# B&R Automation Studio project CleanChemi_SiteManagementSystem (part 26)

```iecst
		IF gSkid_LR[IdxSkids_LR].VisBool.P101_AUTOCAL_OFF THEN
			gCMD_LR[IdxSkids_LR].Write_P101_AUTOCAL.wP101_AUTOCAL := 1;
			gCMD_LR[IdxSkids_LR].Write_P101_AUTOCAL.Send := TRUE;
			gSkid_LR[IdxSkids_LR].VisBool.P101_AUTOCAL_OFF := FALSE;
		END_IF;

		IF gSkid_LR[IdxSkids_LR].VisBool.P102_AUTOCAL_ON THEN
			gCMD_LR[IdxSkids_LR].Write_P102_AUTOCAL.wP102_AUTOCAL := 2;
			gCMD_LR[IdxSkids_LR].Write_P102_AUTOCAL.Send := TRUE;
			gSkid_LR[IdxSkids_LR].VisBool.P102_AUTOCAL_ON := FALSE;
		END_IF;

		IF gSkid_LR[IdxSkids_LR].VisBool.P102_AUTOCAL_OFF THEN
			gCMD_LR[IdxSkids_LR].Write_P102_AUTOCAL.wP102_AUTOCAL := 1;
			gCMD_LR[IdxSkids_LR].Write_P102_AUTOCAL.Send := TRUE;
			gSkid_LR[IdxSkids_LR].VisBool.P102_AUTOCAL_OFF := FALSE;
		END_IF;

		IF gSkid_LR[IdxSkids_LR].VisBool.P103_AUTOCAL_ON THEN
			gCMD_LR[IdxSkids_LR].Write_P103_AUTOCAL.wP103_AUTOCAL := 2;
			gCMD_LR[IdxSkids_LR].Write_P103_AUTOCAL.Send := TRUE;
			gSkid_LR[IdxSkids_LR].VisBool.P103_AUTOCAL_ON := FALSE;
		END_IF;

		IF gSkid_LR[IdxSkids_LR].VisBool.P103_AUTOCAL_OFF THEN
			gCMD_LR[IdxSkids_LR].Write_P103_AUTOCAL.wP103_AUTOCAL := 1;
			gCMD_LR[IdxSkids_LR].Write_P103_AUTOCAL.Send := TRUE;
			gSkid_LR[IdxSkids_LR].VisBool.P103_AUTOCAL_OFF := FALSE;
		END_IF;

		IF gSkid_LR[IdxSkids_LR].VisBool.P104_AUTOCAL_ON THEN
			gCMD_LR[IdxSkids_LR].Write_P104_AUTOCAL.wP104_AUTOCAL := 2;
			gCMD_LR[IdxSkids_LR].Write_P104_AUTOCAL.Send := TRUE;
			gSkid_LR[IdxSkids_LR].VisBool.P104_AUTOCAL_ON := FALSE;
		END_IF;

		IF gSkid_LR[IdxSkids_LR].VisBool.P104_AUTOCAL_OFF THEN
			gCMD_LR[IdxSkids_LR].Write_P104_AUTOCAL.wP104_AUTOCAL := 1;
			gCMD_LR[IdxSkids_LR].Write_P104_AUTOCAL.Send := TRUE;
			gSkid_LR[IdxSkids_LR].VisBool.P104_AUTOCAL_OFF := FALSE;
		END_IF;

		IF gSkid_LR[IdxSkids_LR].VisBool.P201_AUTOCAL_ON THEN
			gCMD_LR[IdxSkids_LR].Write_P201_AUTOCAL.wP201_AUTOCAL := 2;
			gCMD_LR[IdxSkids_LR].Write_P201_AUTOCAL.Send := TRUE;
			gSkid_LR[IdxSkids_LR].VisBool.P201_AUTOCAL_ON := FALSE;
		END_IF;

		IF gSkid_LR[IdxSkids_LR].VisBool.P201_AUTOCAL_OFF THEN
			gCMD_LR[IdxSkids_LR].Write_P201_AUTOCAL.wP201_AUTOCAL := 1;
			gCMD_LR[IdxSkids_LR].Write_P201_AUTOCAL.Send := TRUE;
			gSkid_LR[IdxSkids_LR].VisBool.P201_AUTOCAL_OFF := FALSE;
		END_IF;

		IF gSkid_LR[IdxSkids_LR].VisBool.P202_AUTOCAL_ON THEN
			gCMD_LR[IdxSkids_LR].Write_P202_AUTOCAL.wP202_AUTOCAL := 2;
			gCMD_LR[IdxSkids_LR].Write_P202_AUTOCAL.Send := TRUE;
			gSkid_LR[IdxSkids_LR].VisBool.P202_AUTOCAL_ON := FALSE;
		END_IF;

		IF gSkid_LR[IdxSkids_LR].VisBool.P202_AUTOCAL_OFF THEN
			gCMD_LR[IdxSkids_LR].Write_P202_AUTOCAL.wP202_AUTOCAL := 1;
			gCMD_LR[IdxSkids_LR].Write_P202_AUTOCAL.Send := TRUE;
			gSkid_LR[IdxSkids_LR].VisBool.P202_AUTOCAL_OFF := FALSE;
		END_IF;

		IF gSkid_LR[IdxSkids_LR].VisBool.P203_AUTOCAL_ON THEN
			gCMD_LR[IdxSkids_LR].Write_P203_AUTOCAL.wP203_AUTOCAL := 2;
			gCMD_LR[IdxSkids_LR].Write_P203_AUTOCAL.Send := TRUE;
			gSkid_LR[IdxSkids_LR].VisBool.P203_AUTOCAL_ON := FALSE;
		END_IF;

		IF gSkid_LR[IdxSkids_LR].VisBool.P203_AUTOCAL_OFF THEN
			gCMD_LR[IdxSkids_LR].Write_P203_AUTOCAL.wP203_AUTOCAL := 1;
			gCMD_LR[IdxSkids_LR].Write_P203_AUTOCAL.Send := TRUE;
			gSkid_LR[IdxSkids_LR].VisBool.P203_AUTOCAL_OFF := FALSE;
		END_IF;

		// AutoFLOW 1 = Off, 2 = On
		IF gSkid_LR[IdxSkids_LR].VisBool.P102_AUTOFLOW_ON THEN
			gCMD_LR[IdxSkids_LR].Write_P102_AUTOFLO_ADPT.wP102_P102_AUTOFLO_ADPT := 2;
			gCMD_LR[IdxSkids_LR].Write_P102_AUTOFLO_ADPT.Send := TRUE;
			gSkid_LR[IdxSkids_LR].VisBool.P102_AUTOFLOW_ON := FALSE;
		END_IF;

		IF gSkid_LR[IdxSkids_LR].VisBool.P102_AUTOFLOW_OFF THEN
			gCMD_LR[IdxSkids_LR].Write_P102_AUTOFLO_ADPT.wP102_P102_AUTOFLO_ADPT := 1;
			gCMD_LR[IdxSkids_LR].Write_P102_AUTOFLO_ADPT.Send := TRUE;
			gSkid_LR[IdxSkids_LR].VisBool.P102_AUTOFLOW_OFF := FALSE;
		END_IF;

		IF gSkid_LR[IdxSkids_LR].VisBool.P103_AUTOFLOW_ON THEN
			gCMD_LR[IdxSkids_LR].Write_P103_AUTOFLO_ADPT.wP103_P103_AUTOFLO_ADPT := 2;
			gCMD_LR[IdxSkids_LR].Write_P103_AUTOFLO_ADPT.Send := TRUE;
			gSkid_LR[IdxSkids_LR].VisBool.P103_AUTOFLOW_ON := FALSE;
		END_IF;

		IF gSkid_LR[IdxSkids_LR].VisBool.P103_AUTOFLOW_OFF THEN
			gCMD_LR[IdxSkids_LR].Write_P103_AUTOFLO_ADPT.wP103_P103_AUTOFLO_ADPT := 1;
			gCMD_LR[IdxSkids_LR].Write_P103_AUTOFLO_ADPT.Send := TRUE;
			gSkid_LR[IdxSkids_LR].VisBool.P103_AUTOFLOW_OFF := FALSE;
		END_IF;

		IF gSkid_LR[IdxSkids_LR].VisBool.P104_AUTOFLOW_ON THEN
			gCMD_LR[IdxSkids_LR].Write_P104_AUTOFLO_ADPT.wP104_P104_AUTOFLO_ADPT := 2;
			gCMD_LR[IdxSkids_LR].Write_P104_AUTOFLO_ADPT.Send := TRUE;
			gSkid_LR[IdxSkids_LR].VisBool.P104_AUTOFLOW_ON := FALSE;
		END_IF;

		IF gSkid_LR[IdxSkids_LR].VisBool.P104_AUTOFLOW_OFF THEN
			gCMD_LR[IdxSkids_LR].Write_P104_AUTOFLO_ADPT.wP104_P104_AUTOFLO_ADPT := 1;
			gCMD_LR[IdxSkids_LR].Write_P104_AUTOFLO_ADPT.Send := TRUE;
			gSkid_LR[IdxSkids_LR].VisBool.P104_AUTOFLOW_OFF := FALSE;
		END_IF;

		IF gSkid_LR[IdxSkids_LR].VisBool.P201_AUTOFLOW_ON THEN
			gCMD_LR[IdxSkids_LR].Write_P201_AUTOFLO_ADPT.wP201_P201_AUTOFLO_ADPT := 2;
			gCMD_LR[IdxSkids_LR].Write_P201_AUTOFLO_ADPT.Send := TRUE;
			gSkid_LR[IdxSkids_LR].VisBool.P201_AUTOFLOW_ON := FALSE;
		END_IF;

		IF gSkid_LR[IdxSkids_LR].VisBool.P201_AUTOFLOW_OFF THEN
			gCMD_LR[IdxSkids_LR].Write_P201_AUTOFLO_ADPT.wP201_P201_AUTOFLO_ADPT := 1;
			gCMD_LR[IdxSkids_LR].Write_P201_AUTOFLO_ADPT.Send := TRUE;
			gSkid_LR[IdxSkids_LR].VisBool.P201_AUTOFLOW_OFF := FALSE;
		END_IF;

		IF gSkid_LR[IdxSkids_LR].VisBool.P202_AUTOFLOW_ON THEN
			gCMD_LR[IdxSkids_LR].Write_P202_AUTOFLO_ADPT.wP202_P202_AUTOFLO_ADPT := 2;
			gCMD_LR[IdxSkids_LR].Write_P202_AUTOFLO_ADPT.Send := TRUE;
			gSkid_LR[IdxSkids_LR].VisBool.P202_AUTOFLOW_ON := FALSE;
		END_IF;

		IF gSkid_LR[IdxSkids_LR].VisBool.P202_AUTOFLOW_OFF THEN
			gCMD_LR[IdxSkids_LR].Write_P202_AUTOFLO_ADPT.wP202_P202_AUTOFLO_ADPT := 1;
			gCMD_LR[IdxSkids_LR].Write_P202_AUTOFLO_ADPT.Send := TRUE;
			gSkid_LR[IdxSkids_LR].VisBool.P202_AUTOFLOW_OFF := FALSE;
		END_IF;

		IF gSkid_LR[IdxSkids_LR].VisBool.P203_AUTOFLOW_ON THEN
			gCMD_LR[IdxSkids_LR].Write_P203_AUTOFLO_ADPT.wP203_P203_AUTOFLO_ADPT := 2;
			gCMD_LR[IdxSkids_LR].Write_P203_AUTOFLO_ADPT.Send := TRUE;
			gSkid_LR[IdxSkids_LR].VisBool.P203_AUTOFLOW_ON := FALSE;
		END_IF;

		IF gSkid_LR[IdxSkids_LR].VisBool.P203_AUTOFLOW_OFF THEN
			gCMD_LR[IdxSkids_LR].Write_P203_AUTOFLO_ADPT.wP203_P203_AUTOFLO_ADPT := 1;
			gCMD_LR[IdxSkids_LR].Write_P203_AUTOFLO_ADPT.Send := TRUE;
			gSkid_LR[IdxSkids_LR].VisBool.P203_AUTOFLOW_OFF := FALSE;
		END_IF;

		// Autocal PV 1 = FIT, 2 = PFIT
		IF gSkid_LR[IdxSkids_LR].VisBool.P104_PV_FIT THEN
			gCMD_LR[IdxSkids_LR].Write_P104_AUTOCAL_PV.wP104_AUTOCAL_PV := 1;
			gCMD_LR[IdxSkids_LR].Write_P104_AUTOCAL_PV.Send := TRUE;
			gSkid_LR[IdxSkids_LR].VisBool.P104_PV_FIT := FALSE;
		END_IF;

		IF gSkid_LR[IdxSkids_LR].VisBool.P104_PV_PFIT THEN
			gCMD_LR[IdxSkids_LR].Write_P104_AUTOCAL_PV.wP104_AUTOCAL_PV := 2;
			gCMD_LR[IdxSkids_LR].Write_P104_AUTOCAL_PV.Send := TRUE;
			gSkid_LR[IdxSkids_LR].VisBool.P104_PV_PFIT := FALSE;
		END_IF;

		IF gSkid_LR[IdxSkids_LR].VisBool.P201_PV_FIT THEN
			gCMD_LR[IdxSkids_LR].Write_P201_AUTOCAL_PV.wP201_AUTOCAL_PV := 1;
			gCMD_LR[IdxSkids_LR].Write_P201_AUTOCAL_PV.Send := TRUE;
			gSkid_LR[IdxSkids_LR].VisBool.P201_PV_FIT := FALSE;
		END_IF;

		IF gSkid_LR[IdxSkids_LR].VisBool.P201_PV_PFIT THEN
			gCMD_LR[IdxSkids_LR].Write_P201_AUTOCAL_PV.wP201_AUTOCAL_PV := 2;
			gCMD_LR[IdxSkids_LR].Write_P201_AUTOCAL_PV.Send := TRUE;
			gSkid_LR[IdxSkids_LR].VisBool.P201_PV_PFIT := FALSE;
		END_IF;

		IF gSkid_LR[IdxSkids_LR].VisBool.P202_PV_FIT THEN
			gCMD_LR[IdxSkids_LR].Write_P202_AUTOCAL_PV.wP202_AUTOCAL_PV := 1;
			gCMD_LR[IdxSkids_LR].Write_P202_AUTOCAL_PV.Send := TRUE;
			gSkid_LR[IdxSkids_LR].VisBool.P202_PV_FIT := FALSE;
		END_IF;

		IF gSkid_LR[IdxSkids_LR].VisBool.P202_PV_PFIT THEN
			gCMD_LR[IdxSkids_LR].Write_P202_AUTOCAL_PV.wP202_AUTOCAL_PV := 2;
			gCMD_LR[IdxSkids_LR].Write_P202_AUTOCAL_PV.Send := TRUE;
			gSkid_LR[IdxSkids_LR].VisBool.P202_PV_PFIT := FALSE;
		END_IF;

		IF gSkid_LR[IdxSkids_LR].VisBool.P203_PV_FIT THEN
			gCMD_LR[IdxSkids_LR].Write_P203_AUTOCAL_PV.wP203_AUTOCAL_PV := 1;
			gCMD_LR[IdxSkids_LR].Write_P203_AUTOCAL_PV.Send := TRUE;
			gSkid_LR[IdxSkids_LR].VisBool.P203_PV_FIT := FALSE;
		END_IF;

		IF gSkid_LR[IdxSkids_LR].VisBool.P203_PV_PFIT THEN
			gCMD_LR[IdxSkids_LR].Write_P203_AUTOCAL_PV.wP203_AUTOCAL_PV := 2;
			gCMD_LR[IdxSkids_LR].Write_P203_AUTOCAL_PV.Send := TRUE;
			gSkid_LR[IdxSkids_LR].VisBool.P203_PV_PFIT := FALSE;
		END_IF;

		gSkid_LR[IdxSkids_LR].BufferTank.LI200P := (gSkid_LR[IdxSkids_LR].BufferTank.LI200 / BT_VOLUME)*100;

		gSkid_LR[IdxSkids_LR].VisBool.CD101_TARGETHI := gSkid_LR[IdxSkids_LR].Sensor_Variables.CD101_SP + 40;
		gSkid_LR[IdxSkids_LR].VisBool.CD101_TARGETLO := gSkid_LR[IdxSkids_LR].Sensor_Variables.CD101_SP - 40;
		gSkid_LR[IdxSkids_LR].VisBool.CD102_TARGETHI := gSkid_LR[IdxSkids_LR].Sensor_Variables.CD102_SP + 40;
		gSkid_LR[IdxSkids_LR].VisBool.CD102_TARGETLO := gSkid_LR[IdxSkids_LR].Sensor_Variables.CD102_SP - 40;

		// VISIBILITY TRIGGER SETTING

		IF gSkid_LR[IdxSkids_LR].BufferTank.LSHH200 > LSHH200_TRIGGER THEN
			gSkid_LR[IdxSkids_LR].VisBool.LSHH200 := 1;
		ELSE
			gSkid_LR[IdxSkids_LR].VisBool.LSHH200 := 0;
		END_IF;

		IF gSkid_LR[IdxSkids_LR].Pmax_Pump_102.P102_LS > P102_LS_TRIGGER THEN
			gSkid_LR[IdxSkids_LR].VisBool.P102_LS := 1;
		ELSE
			gSkid_LR[IdxSkids_LR].VisBool.P102_LS := 0;
		END_IF;

		IF gSkid_LR[IdxSkids_LR].Pmax_Pump_103.P103_LS > P103_LS_TRIGGER THEN
			gSkid_LR[IdxSkids_LR].VisBool.P103_LS := 1;
		ELSE
			gSkid_LR[IdxSkids_LR].VisBool.P103_LS := 0;
		END_IF;

		IF gSkid_LR[IdxSkids_LR].Pmax_General_Variables.PMAX_HOA = 2 THEN
			gSkid_LR[IdxSkids_LR].VisBool.PMAX_MANUAL := 1;
		ELSE
			gSkid_LR[IdxSkids_LR].VisBool.PMAX_MANUAL := 0;
		END_IF;

		IF gSkid_LR[IdxSkids_LR].Dosing_Pump_201.P201_HOA = 0 OR gSkid_LR[IdxSkids_LR].Dosing_Pump_201.P201_HOA = 8  THEN
			gSkid_LR[IdxSkids_LR].VisBool.P201_PPM := 0;
		ELSE
			gSkid_LR[IdxSkids_LR].VisBool.P201_PPM := 1;
		END_IF;

		IF gSkid_LR[IdxSkids_LR].Dosing_Pump_202.P202_HOA = 0 OR gSkid_LR[IdxSkids_LR].Dosing_Pump_202.P202_HOA = 8  THEN
			gSkid_LR[IdxSkids_LR].VisBool.P202_PPM := 0;
		ELSE
			gSkid_LR[IdxSkids_LR].VisBool.P202_PPM := 1;
		END_IF;

		IF gSkid_LR[IdxSkids_LR].Dosing_Pump_203.P203_HOA = 0 OR gSkid_LR[IdxSkids_LR].Dosing_Pump_203.P203_HOA = 8  THEN
			gSkid_LR[IdxSkids_LR].VisBool.P203_PPM := 0;
		ELSE
			gSkid_LR[IdxSkids_LR].VisBool.P203_PPM := 1;
		END_IF;

		IF gSkid_LR[IdxSkids_LR].Dosing_Pump_201.P201_HOA = 8 THEN
			gSkid_LR[IdxSkids_LR].VisBool.P201_SP := 1;
		ELSE
			gSkid_LR[IdxSkids_LR].VisBool.P201_SP := 0;
		END_IF;

		IF gSkid_LR[IdxSkids_LR].Dosing_Pump_202.P202_HOA = 8 THEN
			gSkid_LR[IdxSkids_LR].VisBool.P202_SP := 1;
		ELSE
			gSkid_LR[IdxSkids_LR].VisBool.P202_SP := 0;
		END_IF;

		IF gSkid_LR[IdxSkids_LR].Dosing_Pump_203.P203_HOA = 8 THEN
			gSkid_LR[IdxSkids_LR].VisBool.P203_SP := 1;
		ELSE
			gSkid_LR[IdxSkids_LR].VisBool.P203_SP := 0;
		END_IF;

		IF gSkid_LR[IdxSkids_LR].Dosing_Pump_201.P201_ENABLE = 1 THEN
			gSkid_LR[IdxSkids_LR].VisBool.P201_ENABLE_OPP := 0;
		ELSE
			gSkid_LR[IdxSkids_LR].VisBool.P201_ENABLE_OPP := 1;
		END_IF;

		IF gSkid_LR[IdxSkids_LR].Dosing_Pump_202.P202_ENABLE = 1 THEN
			gSkid_LR[IdxSkids_LR].VisBool.P202_ENABLE_OPP := 0;
		ELSE
			gSkid_LR[IdxSkids_LR].VisBool.P202_ENABLE_OPP := 1;
		END_IF;

		IF gSkid_LR[IdxSkids_LR].Dosing_Pump_203.P203_ENABLE = 1 THEN
			gSkid_LR[IdxSkids_LR].VisBool.P203_ENABLE_OPP := 0;
		ELSE
			gSkid_LR[IdxSkids_LR].VisBool.P203_ENABLE_OPP := 1;
		END_IF;

		IF gSkid_LR[IdxSkids_LR].Pmax_Pump_102.P102_WARN > 0 THEN
			gSkid_LR[IdxSkids_LR].VisBool.P102_WARN := 1;
		ELSE
			gSkid_LR[IdxSkids_LR].VisBool.P102_WARN := 0;
		END_IF;

		IF gSkid_LR[IdxSkids_LR].Pmax_Pump_102.P102_ALARM > 0 THEN
			gSkid_LR[IdxSkids_LR].VisBool.P102_ALARM := 1;
		ELSE
			gSkid_LR[IdxSkids_LR].VisBool.P102_ALARM := 0;
		END_IF;

		IF gSkid_LR[IdxSkids_LR].Pmax_Pump_103.P103_WARN > 0 THEN
			gSkid_LR[IdxSkids_LR].VisBool.P103_WARN := 1;
		ELSE
			gSkid_LR[IdxSkids_LR].VisBool.P103_WARN := 0;
		END_IF;

		IF gSkid_LR[IdxSkids_LR].Pmax_Pump_103.P103_ALARM > 0 THEN
			gSkid_LR[IdxSkids_LR].VisBool.P103_ALARM := 1;
		ELSE
			gSkid_LR[IdxSkids_LR].VisBool.P103_ALARM := 0;
		END_IF;

		IF gSkid_LR[IdxSkids_LR].Pmax_Pump_104.P104_WARN > 0 THEN
			gSkid_LR[IdxSkids_LR].VisBool.P104_WARN := 1;
		ELSE
			gSkid_LR[IdxSkids_LR].VisBool.P104_WARN := 0;
		END_IF;

		IF gSkid_LR[IdxSkids_LR].Pmax_Pump_104.P104_ALARM > 0 THEN
			gSkid_LR[IdxSkids_LR].VisBool.P104_ALARM := 1;
		ELSE
			gSkid_LR[IdxSkids_LR].VisBool.P104_ALARM := 0;
		END_IF;

		IF gSkid_LR[IdxSkids_LR].Dosing_Pump_201.P201_WARN > 0 AND gSkid_LR[IdxSkids_LR].VisBool.P201_DME = 0 THEN
			gSkid_LR[IdxSkids_LR].VisBool.P201_WARN := 1;
		ELSE
			gSkid_LR[IdxSkids_LR].VisBool.P201_WARN := 0;
		END_IF;

		IF gSkid_LR[IdxSkids_LR].Dosing_Pump_201.P201_ALARM > 0 AND gSkid_LR[IdxSkids_LR].VisBool.P201_DME = 0  THEN
			gSkid_LR[IdxSkids_LR].VisBool.P201_ALARM := 1;
		ELSE
			gSkid_LR[IdxSkids_LR].VisBool.P201_ALARM := 0;
		END_IF;

		IF gSkid_LR[IdxSkids_LR].Dosing_Pump_202.P202_WARN > 0 THEN
			gSkid_LR[IdxSkids_LR].VisBool.P202_WARN := 1;
		ELSE
			gSkid_LR[IdxSkids_LR].VisBool.P202_WARN := 0;
		END_IF;

		IF gSkid_LR[IdxSkids_LR].Dosing_Pump_202.P202_ALARM > 0 THEN
			gSkid_LR[IdxSkids_LR].VisBool.P202_ALARM := 1;
		ELSE
			gSkid_LR[IdxSkids_LR].VisBool.P202_ALARM := 0;
		END_IF;

		IF gSkid_LR[IdxSkids_LR].Dosing_Pump_203.P203_WARN > 0 THEN
			gSkid_LR[IdxSkids_LR].VisBool.P203_WARN := 1;
		ELSE
			gSkid_LR[IdxSkids_LR].VisBool.P203_WARN := 0;
		END_IF;

		IF gSkid_LR[IdxSkids_LR].Dosing_Pump_203.P203_ALARM > 0 THEN
			gSkid_LR[IdxSkids_LR].VisBool.P203_ALARM := 1;
		ELSE
			gSkid_LR[IdxSkids_LR].VisBool.P203_ALARM := 0;
		END_IF;

		IF gSkid_LR[IdxSkids_LR].Dosing_Pump_201.P201_ADJ = 1 AND gSkid_LR[IdxSkids_LR].VisBool.P201_PPM = 1 THEN
			gSkid_LR[IdxSkids_LR].VisBool.P201_APPM := 1;
		ELSE
			gSkid_LR[IdxSkids_LR].VisBool.P201_APPM := 0;
		END_IF;

		IF gSkid_LR[IdxSkids_LR].Dosing_Pump_202.P202_ADJ = 1 AND gSkid_LR[IdxSkids_LR].VisBool.P202_PPM = 1 THEN
			gSkid_LR[IdxSkids_LR].VisBool.P202_APPM := 1;
		ELSE
			gSkid_LR[IdxSkids_LR].VisBool.P202_APPM := 0;
		END_IF;

		IF gSkid_LR[IdxSkids_LR].Dosing_Pump_203.P203_ADJ = 1 AND gSkid_LR[IdxSkids_LR].VisBool.P203_PPM = 1 THEN
			gSkid_LR[IdxSkids_LR].VisBool.P203_APPM := 1;
		ELSE
			gSkid_LR[IdxSkids_LR].VisBool.P203_APPM := 0;
		END_IF;

		IF gSkid_LR[IdxSkids_LR].Sensor_Variables.FI301_MODE = 0 AND gSkid_LR[IdxSkids_LR].Pmax_General_Variables.SCREEN_LOCK = 1 THEN
			gSkid_LR[IdxSkids_LR].VisBool.FI301_MODE_OPP := 1;
		ELSE
			gSkid_LR[IdxSkids_LR].VisBool.FI301_MODE_OPP := 0;
		END_IF;

		IF gSkid_LR[IdxSkids_LR].Sensor_Variables.FI302_MODE = 0 AND gSkid_LR[IdxSkids_LR].Pmax_General_Variables.SCREEN_LOCK = 1 THEN
			gSkid_LR[IdxSkids_LR].VisBool.FI302_MODE_OPP := 1;
		ELSE
			gSkid_LR[IdxSkids_LR].VisBool.FI302_MODE_OPP := 0;
		END_IF;

		IF gSkid_LR[IdxSkids_LR].Sensor_Variables.FI303_MODE = 0 AND gSkid_LR[IdxSkids_LR].Pmax_General_Variables.SCREEN_LOCK = 1 THEN
			gSkid_LR[IdxSkids_LR].VisBool.FI303_MODE_OPP := 1;
		ELSE
			gSkid_LR[IdxSkids_LR].VisBool.FI303_MODE_OPP := 0;
		END_IF;

		IF gSkid_LR[IdxSkids_LR].Sensor_Variables.FI301_MODE = 1 AND gSkid_LR[IdxSkids_LR].Pmax_General_Variables.SCREEN_LOCK = 1 THEN
			gSkid_LR[IdxSkids_LR].VisBool.FI301_MODE := 1;
		ELSE
			gSkid_LR[IdxSkids_LR].VisBool.FI301_MODE := 0;
		END_IF;

		IF gSkid_LR[IdxSkids_LR].Sensor_Variables.FI302_MODE = 1 AND gSkid_LR[IdxSkids_LR].Pmax_General_Variables.SCREEN_LOCK = 1 THEN
			gSkid_LR[IdxSkids_LR].VisBool.FI302_MODE := 1;
		ELSE
			gSkid_LR[IdxSkids_LR].VisBool.FI302_MODE := 0;
		END_IF;

		IF gSkid_LR[IdxSkids_LR].Sensor_Variables.FI303_MODE = 1 AND gSkid_LR[IdxSkids_LR].Pmax_General_Variables.SCREEN_LOCK = 1 THEN
			gSkid_LR[IdxSkids_LR].VisBool.FI303_MODE := 1;
		ELSE
			gSkid_LR[IdxSkids_LR].VisBool.FI303_MODE := 0;
		END_IF;

		IF gSkid_LR[IdxSkids_LR].Sensor_Variables.XV101 = 0 AND gSkid_LR[IdxSkids_LR].Sensor_Variables.XV101_ENABLE = 1 THEN
			gSkid_LR[IdxSkids_LR].VisBool.XV101_OPP := 1;
		ELSE
			gSkid_LR[IdxSkids_LR].VisBool.XV101_OPP := 0;
		END_IF;

		IF gSkid_LR[IdxSkids_LR].Sensor_Variables.XV101 = 2 AND gSkid_LR[IdxSkids_LR].Sensor_Variables.XV101_ENABLE = 1 THEN
			gSkid_LR[IdxSkids_LR].VisBool.XV101_ERROR := 1;
		ELSE
			gSkid_LR[IdxSkids_LR].VisBool.XV101_ERROR := 0;
		END_IF;

		IF gSkid_LR[IdxSkids_LR].Sensor_Variables.XV101 = 1 AND gSkid_LR[IdxSkids_LR].Sensor_Variables.XV101_ENABLE = 1 THEN
			gSkid_LR[IdxSkids_LR].VisBool.XV101 := 1;
		ELSE
			gSkid_LR[IdxSkids_LR].VisBool.XV101 := 0;
		END_IF;

		IF gSkid_LR[IdxSkids_LR].Sensor_Variables.XV102 = 0 AND gSkid_LR[IdxSkids_LR].Pmax_Pump_102.XV102_ENABLE = 1 THEN
			gSkid_LR[IdxSkids_LR].VisBool.XV102_OPP := 1;
		ELSE
			gSkid_LR[IdxSkids_LR].VisBool.XV102_OPP := 0;
		END_IF;

		IF gSkid_LR[IdxSkids_LR].Sensor_Variables.XV102 = 1 AND gSkid_LR[IdxSkids_LR].Pmax_Pump_102.XV102_ENABLE = 1 THEN
			gSkid_LR[IdxSkids_LR].VisBool.XV102 := 1;
		ELSE
			gSkid_LR[IdxSkids_LR].VisBool.XV102 := 0;
		END_IF;

		IF gSkid_LR[IdxSkids_LR].Sensor_Variables.XV103 = 1 THEN
			gSkid_LR[IdxSkids_LR].VisBool.XV103_OPP := 0;
		ELSE
			gSkid_LR[IdxSkids_LR].VisBool.XV103_OPP := 1;
		END_IF;

		IF gSkid_LR[IdxSkids_LR].Sensor_Variables.XV104 = 0 AND gSkid_LR[IdxSkids_LR].Pmax_Pump_104.XV104_ENABLE = 1 THEN
			gSkid_LR[IdxSkids_LR].VisBool.XV104_OPP := 1;
		ELSE
			gSkid_LR[IdxSkids_LR].VisBool.XV104_OPP := 0;
		END_IF;

		IF gSkid_LR[IdxSkids_LR].Sensor_Variables.XV104 = 1 AND gSkid_LR[IdxSkids_LR].Pmax_Pump_104.XV104_ENABLE = 1 THEN
			gSkid_LR[IdxSkids_LR].VisBool.XV104 := 1;
		ELSE
			gSkid_LR[IdxSkids_LR].VisBool.XV104 := 0;
		END_IF;

		IF gSkid_LR[IdxSkids_LR].Sensor_Variables.XV201 = 1 THEN
			gSkid_LR[IdxSkids_LR].VisBool.XV201_OPP := 0;
		ELSE
			gSkid_LR[IdxSkids_LR].VisBool.XV201_OPP := 1;
		END_IF;

		IF gSkid_LR[IdxSkids_LR].Sensor_Variables.XV202 = 1 THEN
			gSkid_LR[IdxSkids_LR].VisBool.XV202_OPP := 0;
		ELSE
			gSkid_LR[IdxSkids_LR].VisBool.XV202_OPP := 1;
		END_IF;

		IF gSkid_LR[IdxSkids_LR].Sensor_Variables.XV203 = 1 THEN
			gSkid_LR[IdxSkids_LR].VisBool.XV203_OPP := 0;
		ELSE
			gSkid_LR[IdxSkids_LR].VisBool.XV203_OPP := 1;
		END_IF;

		IF gSkid_LR[IdxSkids_LR].Dosing_Pump_201.P201_PTYPE = 1 THEN
			gSkid_LR[IdxSkids_LR].VisBool.P201_PTYPE_OPP := 0;
		ELSE
			gSkid_LR[IdxSkids_LR].VisBool.P201_PTYPE_OPP := 1;
		END_IF;

		IF gSkid_LR[IdxSkids_LR].Pmax_General_Variables.SCREEN_LOCK = 1 AND gSkid_LR[IdxSkids_LR].Pmax_General_Variables.PMAX_HOA = 2 THEN
			gSkid_LR[IdxSkids_LR].VisBool.P101_MODE := 1;
			gSkid_LR[IdxSkids_LR].VisBool.P102_MODE := 1;
			gSkid_LR[IdxSkids_LR].VisBool.P103_MODE := 1;
			gSkid_LR[IdxSkids_LR].VisBool.P104_MODE := 1;
		ELSE
			gSkid_LR[IdxSkids_LR].VisBool.P101_MODE := 0;
			gSkid_LR[IdxSkids_LR].VisBool.P102_MODE := 0;
			gSkid_LR[IdxSkids_LR].VisBool.P103_MODE := 0;
			gSkid_LR[IdxSkids_LR].VisBool.P104_MODE := 0;
		END_IF;

		IF gSkid_LR[IdxSkids_LR].Pmax_General_Variables.SCREEN_LOCK = 1 AND gSkid_LR[IdxSkids_LR].Dosing_Pump_201.P201_HOA = 8 THEN
			gSkid_LR[IdxSkids_LR].VisBool.P201_MODE := 1;
		ELSE
			gSkid_LR[IdxSkids_LR].VisBool.P201_MODE := 0;
		END_IF;

		IF gSkid_LR[IdxSkids_LR].Pmax_General_Variables.SCREEN_LOCK = 1 AND gSkid_LR[IdxSkids_LR].Dosing_Pump_202.P202_HOA = 8 THEN
			gSkid_LR[IdxSkids_LR].VisBool.P202_MODE := 1;
		ELSE
			gSkid_LR[IdxSkids_LR].VisBool.P202_MODE := 0;
		END_IF;

		IF gSkid_LR[IdxSkids_LR].Pmax_General_Variables.SCREEN_LOCK = 1 AND gSkid_LR[IdxSkids_LR].Dosing_Pump_203.P203_HOA = 8 THEN
			gSkid_LR[IdxSkids_LR].VisBool.P203_MODE := 1;
		ELSE
			gSkid_LR[IdxSkids_LR].VisBool.P203_MODE := 0;
		END_IF;

		IF gSkid_LR[IdxSkids_LR].Heartbeat.SYSTEM_OFFLINE = 1 THEN
			gSkid_LR[IdxSkids_LR].VisBool.IOSTATUS := 1;
		ELSE
			gSkid_LR[IdxSkids_LR].VisBool.IOSTATUS := 0;
		END_IF;

		//P101 Pump Graphic Vis
		IF gSkid_LR[IdxSkids_LR].Pmax_Pump_101.P101_XS = 1 THEN
			gSkid_LR[IdxSkids_LR].VisBool.P101_DMEYELLOW := 1;
		ELSE
			gSkid_LR[IdxSkids_LR].VisBool.P101_DMEYELLOW := 0;
		END_IF;

		IF gSkid_LR[IdxSkids_LR].Pmax_Pump_101.P101_XS = 3 THEN
			gSkid_LR[IdxSkids_LR].VisBool.P101_DMEGREEN := 1;
		ELSE
			gSkid_LR[IdxSkids_LR].VisBool.P101_DMEGREEN := 0;
		END_IF;

		//P102 Pump Graphic Vis
		IF gSkid_LR[IdxSkids_LR].Pmax_Pump_102.P102_XS = 1 THEN
			gSkid_LR[IdxSkids_LR].VisBool.P102_DDAYELLOW := 1;
		ELSE
			gSkid_LR[IdxSkids_LR].VisBool.P102_DDAYELLOW := 0;
		END_IF;

		IF gSkid_LR[IdxSkids_LR].Pmax_Pump_102.P102_XS = 3 THEN
			gSkid_LR[IdxSkids_LR].VisBool.P102_DDAGREEN := 1;
		ELSE
			gSkid_LR[IdxSkids_LR].VisBool.P102_DDAGREEN := 0;
		END_IF;

		//P103 Pump Graphic Vis
		IF gSkid_LR[IdxSkids_LR].Pmax_Pump_103.P103_XS = 1 THEN
			gSkid_LR[IdxSkids_LR].VisBool.P103_DDAYELLOW := 1;
		ELSE
			gSkid_LR[IdxSkids_LR].VisBool.P103_DDAYELLOW := 0;
		END_IF;

		IF gSkid_LR[IdxSkids_LR].Pmax_Pump_103.P103_XS = 3 THEN
			gSkid_LR[IdxSkids_LR].VisBool.P103_DDAGREEN := 1;
		ELSE
			gSkid_LR[IdxSkids_LR].VisBool.P103_DDAGREEN := 0;
		END_IF;

		//P104 Pump Graphic Vis
		IF gSkid_LR[IdxSkids_LR].Pmax_Pump_104.P104_XS = 1 THEN
			gSkid_LR[IdxSkids_LR].VisBool.P104_DDAYELLOW := 1;
		ELSE
			gSkid_LR[IdxSkids_LR].VisBool.P104_DDAYELLOW := 0;
		END_IF;

		IF gSkid_LR[IdxSkids_LR].Pmax_Pump_104.P104_XS = 3 THEN
			gSkid_LR[IdxSkids_LR].VisBool.P104_DDAGREEN := 1;
		ELSE
			gSkid_LR[IdxSkids_LR].VisBool.P104_DDAGREEN := 0;
		END_IF;

		//P201 Pump Graphic Vis
		IF gSkid_LR[IdxSkids_LR].Dosing_Pump_201.P201_PTYPE = 0 THEN
			gSkid_LR[IdxSkids_LR].VisBool.P201_DDA := 1;
			gSkid_LR[IdxSkids_LR].VisBool.P201_DME := 0;
		ELSE
			gSkid_LR[IdxSkids_LR].VisBool.P201_DDA := 0;
			gSkid_LR[IdxSkids_LR].VisBool.P201_DME := 1;
		END_IF;

		IF gSkid_LR[IdxSkids_LR].Dosing_Pump_201.P201_PTYPE = 1 AND gSkid_LR[IdxSkids_LR].Dosing_Pump_201.P201_XS = 3 THEN
			gSkid_LR[IdxSkids_LR].VisBool.P201_DMEGREEN := 1;
		ELSE
			gSkid_LR[IdxSkids_LR].VisBool.P201_DMEGREEN := 0;
		END_IF;

		IF gSkid_LR[IdxSkids_LR].Dosing_Pump_201.P201_PTYPE = 1 AND gSkid_LR[IdxSkids_LR].Dosing_Pump_201.P201_XS = 1 THEN
			gSkid_LR[IdxSkids_LR].VisBool.P201_DMEYELLOW := 1;
		ELSE
			gSkid_LR[IdxSkids_LR].VisBool.P201_DMEYELLOW := 0;
		END_IF;

		IF gSkid_LR[IdxSkids_LR].Dosing_Pump_201.P201_XS = 1 AND gSkid_LR[IdxSkids_LR].Dosing_Pump_201.P201_PTYPE = 0 THEN
			gSkid_LR[IdxSkids_LR].VisBool.P201_DDAYELLOW := 1;
		ELSE
			gSkid_LR[IdxSkids_LR].VisBool.P201_DDAYELLOW := 0;
		END_IF;

		IF gSkid_LR[IdxSkids_LR].Dosing_Pump_201.P201_XS = 3 AND gSkid_LR[IdxSkids_LR].Dosing_Pump_201.P201_PTYPE = 0 THEN
			gSkid_LR[IdxSkids_LR].VisBool.P201_DDAGREEN := 1;
		ELSE
			gSkid_LR[IdxSkids_LR].VisBool.P201_DDAGREEN := 0;
		END_IF;

		//P202 Pump Graphic Vis
		IF gSkid_LR[IdxSkids_LR].Dosing_Pump_202.P202_XS = 1 THEN
			gSkid_LR[IdxSkids_LR].VisBool.P202_DDAYELLOW := 1;
		ELSE
			gSkid_LR[IdxSkids_LR].VisBool.P202_DDAYELLOW := 0;
		END_IF;

		IF gSkid_LR[IdxSkids_LR].Dosing_Pump_202.P202_XS = 3 THEN
			gSkid_LR[IdxSkids_LR].VisBool.P202_DDAGREEN := 1;
		ELSE
			gSkid_LR[IdxSkids_LR].VisBool.P202_DDAGREEN := 0;
		END_IF;

		//P203 Pump Graphic Vis
		IF gSkid_LR[IdxSkids_LR].Dosing_Pump_203.P203_XS = 1 THEN
			gSkid_LR[IdxSkids_LR].VisBool.P203_DDAYELLOW := 1;
		ELSE
			gSkid_LR[IdxSkids_LR].VisBool.P203_DDAYELLOW := 0;
		END_IF;

		IF gSkid_LR[IdxSkids_LR].Dosing_Pump_203.P203_XS = 3 THEN
			gSkid_LR[IdxSkids_LR].VisBool.P203_DDAGREEN := 1;
		ELSE
			gSkid_LR[IdxSkids_LR].VisBool.P203_DDAGREEN := 0;
		END_IF;

	END_FOR;

END_ACTION
```

#### Main_HR.st
```iecst
ACTION Vis_Main_HR:

	FOR IdxSkids_HR := 0 TO MAX_SKIDS_HR DO

		gSkid_HR[IdxSkids_HR].BufferTank.LI200P := (gSkid_HR[IdxSkids_HR].BufferTank.LI200 / BT_VOLUME)*100;

		// VISIBILITY TRIGGER SETTING

		IF gSkid_LR[IdxSkids_HR].Pmax_General_Variables.HEARTBEAT = 1 THEN
			gSkid_LR[IdxSkids_HR].VisBool.HEARTBEAT := 0;
		ELSE
			gSkid_LR[IdxSkids_HR].VisBool.HEARTBEAT := 1;
		END_IF;

		IF gSkid_HR[IdxSkids_HR].BufferTank.LSHH200 > LSHH200_TRIGGER THEN
			gSkid_HR[IdxSkids_HR].VisBool.LSHH200 := 1;
		ELSE
			gSkid_HR[IdxSkids_HR].VisBool.LSHH200 := 0;
		END_IF;

		IF gSkid_HR[IdxSkids_HR].Pmax_Pump_102.P102_LS > P102_LS_TRIGGER THEN
			gSkid_HR[IdxSkids_HR].VisBool.P102_LS := 1;
		ELSE
			gSkid_HR[IdxSkids_HR].VisBool.P102_LS := 0;
		END_IF;

		IF gSkid_HR[IdxSkids_HR].Pmax_Pump_103.P103_LS > P103_LS_TRIGGER THEN
			gSkid_HR[IdxSkids_HR].VisBool.P103_LS := 1;
		ELSE
			gSkid_HR[IdxSkids_HR].VisBool.P103_LS := 0;
		END_IF;

		IF gSkid_HR[IdxSkids_HR].Pmax_General_Variables.PMAX_HOA = 2 THEN
			gSkid_HR[IdxSkids_HR].VisBool.PMAX_MANUAL := 1;
		ELSE
			gSkid_HR[IdxSkids_HR].VisBool.PMAX_MANUAL := 0;
		END_IF;

		IF gSkid_HR[IdxSkids_HR].Dosing_Pump_201.P201_HOA = 0 OR gSkid_HR[IdxSkids_HR].Dosing_Pump_201.P201_HOA = 8  THEN
			gSkid_HR[IdxSkids_HR].VisBool.P201_PPM := 0;
		ELSE
			gSkid_HR[IdxSkids_HR].VisBool.P201_PPM := 1;
		END_IF;

		IF gSkid_HR[IdxSkids_HR].Dosing_Pump_202.P202_HOA = 0 OR gSkid_HR[IdxSkids_HR].Dosing_Pump_202.P202_HOA = 8  THEN
			gSkid_HR[IdxSkids_HR].VisBool.P202_PPM := 0;
		ELSE
			gSkid_HR[IdxSkids_HR].VisBool.P202_PPM := 1;
		END_IF;

		IF gSkid_HR[IdxSkids_HR].Dosing_Pump_203.P203_HOA = 0 OR gSkid_HR[IdxSkids_HR].Dosing_Pump_203.P203_HOA = 8  THEN
			gSkid_HR[IdxSkids_HR].VisBool.P203_PPM := 0;
		ELSE
			gSkid_HR[IdxSkids_HR].VisBool.P203_PPM := 1;
		END_IF;

		IF gSkid_HR[IdxSkids_HR].Dosing_Pump_204.P204_HOA = 0 OR gSkid_HR[IdxSkids_HR].Dosing_Pump_204.P204_HOA = 8  THEN
			gSkid_HR[IdxSkids_HR].VisBool.P204_PPM := 0;
		ELSE
			gSkid_HR[IdxSkids_HR].VisBool.P204_PPM := 1;
		END_IF;

		IF gSkid_HR[IdxSkids_HR].Dosing_Pump_201.P201_HOA = 8 THEN
			gSkid_HR[IdxSkids_HR].VisBool.P201_SP := 1;
		ELSE
			gSkid_HR[IdxSkids_HR].VisBool.P201_SP := 0;
		END_IF;

		IF gSkid_HR[IdxSkids_HR].Dosing_Pump_202.P202_HOA = 8 THEN
			gSkid_HR[IdxSkids_HR].VisBool.P202_SP := 1;
		ELSE
			gSkid_HR[IdxSkids_HR].VisBool.P202_SP := 0;
		END_IF;

		IF gSkid_HR[IdxSkids_HR].Dosing_Pump_203.P203_HOA = 8 THEN
			gSkid_HR[IdxSkids_HR].VisBool.P203_SP := 1;
		ELSE
			gSkid_HR[IdxSkids_HR].VisBool.P203_SP := 0;
		END_IF;

		IF gSkid_HR[IdxSkids_HR].Dosing_Pump_204.P204_HOA = 8 THEN
			gSkid_HR[IdxSkids_HR].VisBool.P204_SP := 1;
		ELSE
			gSkid_HR[IdxSkids_HR].VisBool.P204_SP := 0;
		END_IF;

		IF gSkid_HR[IdxSkids_HR].Dosing_Pump_201.P201_ENABLE = 1 THEN
			gSkid_HR[IdxSkids_HR].VisBool.P201_ENABLE_OPP := 0;
		ELSE
			gSkid_HR[IdxSkids_HR].VisBool.P201_ENABLE_OPP := 1;
		END_IF;

		IF gSkid_HR[IdxSkids_HR].Dosing_Pump_202.P202_ENABLE = 1 THEN
			gSkid_HR[IdxSkids_HR].VisBool.P202_ENABLE_OPP := 0;
		ELSE
			gSkid_HR[IdxSkids_HR].VisBool.P202_ENABLE_OPP := 1;
		END_IF;

		IF gSkid_HR[IdxSkids_HR].Dosing_Pump_203.P203_ENABLE = 1 THEN
			gSkid_HR[IdxSkids_HR].VisBool.P203_ENABLE_OPP := 0;
		ELSE
			gSkid_HR[IdxSkids_HR].VisBool.P203_ENABLE_OPP := 1;
		END_IF;

		IF gSkid_HR[IdxSkids_HR].Dosing_Pump_204.P204_ENABLE = 1 THEN
			gSkid_HR[IdxSkids_HR].VisBool.P204_ENABLE_OPP := 0;
		ELSE
			gSkid_HR[IdxSkids_HR].VisBool.P204_ENABLE_OPP := 1;
		END_IF;

		IF gSkid_HR[IdxSkids_HR].Pmax_Pump_102.P102_WARN > 0 THEN
			gSkid_HR[IdxSkids_HR].VisBool.P102_WARN := 1;
		ELSE
			gSkid_HR[IdxSkids_HR].VisBool.P102_WARN := 0;
		END_IF;

		IF gSkid_HR[IdxSkids_HR].Pmax_Pump_102.P102_ALARM > 0 THEN
			gSkid_HR[IdxSkids_HR].VisBool.P102_ALARM := 1;
		ELSE
			gSkid_HR[IdxSkids_HR].VisBool.P102_ALARM := 0;
		END_IF;

		IF gSkid_HR[IdxSkids_HR].Pmax_Pump_103.P103_WARN > 0 THEN
			gSkid_HR[IdxSkids_HR].VisBool.P103_WARN := 1;
		ELSE
			gSkid_HR[IdxSkids_HR].VisBool.P103_WARN := 0;
		END_IF;

		IF gSkid_HR[IdxSkids_HR].Pmax_Pump_103.P103_ALARM > 0 THEN
			gSkid_HR[IdxSkids_HR].VisBool.P103_ALARM := 1;
		ELSE
			gSkid_HR[IdxSkids_HR].VisBool.P103_ALARM := 0;
		END_IF;

		IF gSkid_HR[IdxSkids_HR].Pmax_Pump_104.P104_WARN > 0 THEN
			gSkid_HR[IdxSkids_HR].VisBool.P104_WARN := 1;
		ELSE
			gSkid_HR[IdxSkids_HR].VisBool.P104_WARN := 0;
		END_IF;

		IF gSkid_HR[IdxSkids_HR].Pmax_Pump_104.P104_ALARM > 0 THEN
			gSkid_HR[IdxSkids_HR].VisBool.P104_ALARM := 1;
		ELSE
			gSkid_HR[IdxSkids_HR].VisBool.P104_ALARM := 0;
		END_IF;

		IF gSkid_HR[IdxSkids_HR].Dosing_Pump_201.P201_WARN > 0 THEN
			gSkid_HR[IdxSkids_HR].VisBool.P201_WARN := 1;
		ELSE
			gSkid_HR[IdxSkids_HR].VisBool.P201_WARN := 0;
		END_IF;

		IF gSkid_HR[IdxSkids_HR].Dosing_Pump_201.P201_ALARM > 0 THEN
			gSkid_HR[IdxSkids_HR].VisBool.P201_ALARM := 1;
		ELSE
			gSkid_HR[IdxSkids_HR].VisBool.P201_ALARM := 0;
		END_IF;

		IF gSkid_HR[IdxSkids_HR].Dosing_Pump_202.P202_WARN > 0 THEN
			gSkid_HR[IdxSkids_HR].VisBool.P202_WARN := 1;
		ELSE
			gSkid_HR[IdxSkids_HR].VisBool.P202_WARN := 0;
		END_IF;

		IF gSkid_HR[IdxSkids_HR].Dosing_Pump_202.P202_ALARM > 0 THEN
			gSkid_HR[IdxSkids_HR].VisBool.P202_ALARM := 1;
		ELSE
			gSkid_HR[IdxSkids_HR].VisBool.P202_ALARM := 0;
		END_IF;

		IF gSkid_HR[IdxSkids_HR].Dosing_Pump_203.P203_WARN > 0 THEN
			gSkid_HR[IdxSkids_HR].VisBool.P203_WARN := 1;
		ELSE
			gSkid_HR[IdxSkids_HR].VisBool.P203_WARN := 0;
		END_IF;

		IF gSkid_HR[IdxSkids_HR].Dosing_Pump_204.P204_WARN > 0 THEN
			gSkid_HR[IdxSkids_HR].VisBool.P204_WARN := 1;
		ELSE
			gSkid_HR[IdxSkids_HR].VisBool.P204_WARN := 0;
		END_IF;

		IF gSkid_HR[IdxSkids_HR].Dosing_Pump_203.P203_ALARM > 0 THEN
			gSkid_HR[IdxSkids_HR].VisBool.P203_ALARM := 1;
		ELSE
			gSkid_HR[IdxSkids_HR].VisBool.P203_ALARM := 0;
		END_IF;

		IF gSkid_HR[IdxSkids_HR].Dosing_Pump_204.P204_ALARM > 0 THEN
			gSkid_HR[IdxSkids_HR].VisBool.P204_ALARM := 1;
		ELSE
			gSkid_HR[IdxSkids_HR].VisBool.P204_ALARM := 0;
		END_IF;

		IF gSkid_HR[IdxSkids_HR].Dosing_Pump_201.P201_ADJ = 1 AND gSkid_HR[IdxSkids_HR].VisBool.P201_PPM = 1 THEN
			gSkid_HR[IdxSkids_HR].VisBool.P201_APPM := 1;
		ELSE
			gSkid_HR[IdxSkids_HR].VisBool.P201_APPM := 0;
		END_IF;

		IF gSkid_HR[IdxSkids_HR].Dosing_Pump_202.P202_ADJ = 1 AND gSkid_HR[IdxSkids_HR].VisBool.P202_PPM = 1 THEN
			gSkid_HR[IdxSkids_HR].VisBool.P202_APPM := 1;
		ELSE
			gSkid_HR[IdxSkids_HR].VisBool.P202_APPM := 0;
		END_IF;

		IF gSkid_HR[IdxSkids_HR].Dosing_Pump_203.P203_ADJ = 1 AND gSkid_HR[IdxSkids_HR].VisBool.P203_PPM = 1 THEN
			gSkid_HR[IdxSkids_HR].VisBool.P203_APPM := 1;
		ELSE
			gSkid_HR[IdxSkids_HR].VisBool.P203_APPM := 0;
		END_IF;

		IF gSkid_HR[IdxSkids_HR].Dosing_Pump_204.P204_ADJ = 1 AND gSkid_HR[IdxSkids_HR].VisBool.P204_PPM = 1 THEN
			gSkid_HR[IdxSkids_HR].VisBool.P204_APPM := 1;
		ELSE
			gSkid_HR[IdxSkids_HR].VisBool.P204_APPM := 0;
		END_IF;

		IF gSkid_HR[IdxSkids_HR].Sensor_Variables.FI301_MODE = 0 AND gSkid_HR[IdxSkids_HR].Pmax_General_Variables.SCREEN_LOCK = 1 THEN
			gSkid_HR[IdxSkids_HR].VisBool.FI301_MODE_OPP := 1;
		ELSE
			gSkid_HR[IdxSkids_HR].VisBool.FI301_MODE_OPP := 0;
		END_IF;

		IF gSkid_HR[IdxSkids_HR].Sensor_Variables.FI302_MODE = 0 AND gSkid_HR[IdxSkids_HR].Pmax_General_Variables.SCREEN_LOCK = 1 THEN
			gSkid_HR[IdxSkids_HR].VisBool.FI302_MODE_OPP := 1;
		ELSE
			gSkid_HR[IdxSkids_HR].VisBool.FI302_MODE_OPP := 0;
		END_IF;

		IF gSkid_HR[IdxSkids_HR].Sensor_Variables.FI303_MODE = 0 AND gSkid_HR[IdxSkids_HR].Pmax_General_Variables.SCREEN_LOCK = 1 THEN
			gSkid_HR[IdxSkids_HR].VisBool.FI303_MODE_OPP := 1;
		ELSE
			gSkid_HR[IdxSkids_HR].VisBool.FI303_MODE_OPP := 0;
		END_IF;

		IF gSkid_HR[IdxSkids_HR].Sensor_Variables.FI304_MODE = 0 AND gSkid_HR[IdxSkids_HR].Pmax_General_Variables.SCREEN_LOCK = 1 THEN
			gSkid_HR[IdxSkids_HR].VisBool.FI304_MODE_OPP := 1;
		ELSE
			gSkid_HR[IdxSkids_HR].VisBool.FI304_MODE_OPP := 0;
		END_IF;

		IF gSkid_HR[IdxSkids_HR].Sensor_Variables.FI301_MODE = 1 AND gSkid_HR[IdxSkids_HR].Pmax_General_Variables.SCREEN_LOCK = 1 THEN
			gSkid_HR[IdxSkids_HR].VisBool.FI301_MODE := 1;
		ELSE
			gSkid_HR[IdxSkids_HR].VisBool.FI301_MODE := 0;
		END_IF;

		IF gSkid_HR[IdxSkids_HR].Sensor_Variables.FI302_MODE = 1 AND gSkid_HR[IdxSkids_HR].Pmax_General_Variables.SCREEN_LOCK = 1 THEN
			gSkid_HR[IdxSkids_HR].VisBool.FI302_MODE := 1;
		ELSE
			gSkid_HR[IdxSkids_HR].VisBool.FI302_MODE := 0;
		END_IF;

		IF gSkid_HR[IdxSkids_HR].Sensor_Variables.FI303_MODE = 1 AND gSkid_HR[IdxSkids_HR].Pmax_General_Variables.SCREEN_LOCK = 1 THEN
			gSkid_HR[IdxSkids_HR].VisBool.FI303_MODE := 1;
		ELSE
			gSkid_HR[IdxSkids_HR].VisBool.FI303_MODE := 0;
		END_IF;

		IF gSkid_HR[IdxSkids_HR].Sensor_Variables.FI304_MODE = 1 AND gSkid_HR[IdxSkids_HR].Pmax_General_Variables.SCREEN_LOCK = 1 THEN
			gSkid_HR[IdxSkids_HR].VisBool.FI304_MODE := 1;
		ELSE
			gSkid_HR[IdxSkids_HR].VisBool.FI304_MODE := 0;
		END_IF;

		IF gSkid_HR[IdxSkids_HR].Sensor_Variables.XV101 = 0 AND gSkid_HR[IdxSkids_HR].Sensor_Variables.XV101_ENABLE = 1 THEN
			gSkid_HR[IdxSkids_HR].VisBool.XV101_OPP := 1;
		ELSE
			gSkid_HR[IdxSkids_HR].VisBool.XV101_OPP := 0;
		END_IF;

		IF gSkid_HR[IdxSkids_HR].Sensor_Variables.XV101 = 1 AND gSkid_HR[IdxSkids_HR].Sensor_Variables.XV101_ENABLE = 1 THEN
			gSkid_HR[IdxSkids_HR].VisBool.XV101 := 1;
		ELSE
			gSkid_HR[IdxSkids_HR].VisBool.XV101 := 0;
		END_IF;

		IF gSkid_HR[IdxSkids_HR].Sensor_Variables.XV102 = 1 THEN
			gSkid_HR[IdxSkids_HR].VisBool.XV102_OPP := 0;
		ELSE
			gSkid_HR[IdxSkids_HR].VisBool.XV102_OPP := 1;
		END_IF;

		IF gSkid_HR[IdxSkids_HR].Sensor_Variables.XV103 = 1 THEN
			gSkid_HR[IdxSkids_HR].VisBool.XV103_OPP := 0;
		ELSE
			gSkid_HR[IdxSkids_HR].VisBool.XV103_OPP := 1;
		END_IF;

		IF gSkid_HR[IdxSkids_HR].Sensor_Variables.XV104 = 1 THEN
			gSkid_HR[IdxSkids_HR].VisBool.XV104_OPP := 0;
		ELSE
			gSkid_HR[IdxSkids_HR].VisBool.XV104_OPP := 1;
		END_IF;

		IF gSkid_HR[IdxSkids_HR].Sensor_Variables.XV201 = 1 THEN
			gSkid_HR[IdxSkids_HR].VisBool.XV201_OPP := 0;
		ELSE
			gSkid_HR[IdxSkids_HR].VisBool.XV201_OPP := 1;
		END_IF;

		IF gSkid_HR[IdxSkids_HR].Sensor_Variables.XV202 = 1 THEN
			gSkid_HR[IdxSkids_HR].VisBool.XV202_OPP := 0;
		ELSE
			gSkid_HR[IdxSkids_HR].VisBool.XV202_OPP := 1;
		END_IF;

		IF gSkid_HR[IdxSkids_HR].Sensor_Variables.XV203 = 1 THEN
			gSkid_HR[IdxSkids_HR].VisBool.XV203_OPP := 0;
		ELSE
			gSkid_HR[IdxSkids_HR].VisBool.XV203_OPP := 1;
		END_IF;

		IF gSkid_HR[IdxSkids_HR].Sensor_Variables.XV204 = 1 THEN
			gSkid_HR[IdxSkids_HR].VisBool.XV204_OPP := 0;
		ELSE
			gSkid_HR[IdxSkids_HR].VisBool.XV204_OPP := 1;
		END_IF;

		IF gSkid_HR[IdxSkids_HR].Dosing_Pump_201.P201_PTYPE = 1 THEN
			gSkid_HR[IdxSkids_HR].VisBool.P201_PTYPE_OPP := 0;
		ELSE
			gSkid_HR[IdxSkids_HR].VisBool.P201_PTYPE_OPP := 1;
		END_IF;

		IF gSkid_HR[IdxSkids_HR].Pmax_General_Variables.SCREEN_LOCK = 1 AND gSkid_HR[IdxSkids_HR].Pmax_General_Variables.PMAX_HOA = 2 THEN
			gSkid_HR[IdxSkids_HR].VisBool.P101_MODE := 1;
			gSkid_HR[IdxSkids_HR].VisBool.P102_MODE := 1;
			gSkid_HR[IdxSkids_HR].VisBool.P103_MODE := 1;
			gSkid_HR[IdxSkids_HR].VisBool.P104_MODE := 1;
		ELSE
			gSkid_HR[IdxSkids_HR].VisBool.P101_MODE := 0;
			gSkid_HR[IdxSkids_HR].VisBool.P102_MODE := 0;
			gSkid_HR[IdxSkids_HR].VisBool.P103_MODE := 0;
			gSkid_HR[IdxSkids_HR].VisBool.P104_MODE := 0;
		END_IF;

		IF gSkid_HR[IdxSkids_HR].Pmax_General_Variables.SCREEN_LOCK = 1 AND gSkid_HR[IdxSkids_HR].Dosing_Pump_201.P201_HOA = 8 THEN
			gSkid_HR[IdxSkids_HR].VisBool.P201_MODE := 1;
		ELSE
			gSkid_HR[IdxSkids_HR].VisBool.P201_MODE := 0;
		END_IF;

		IF gSkid_HR[IdxSkids_HR].Pmax_General_Variables.SCREEN_LOCK = 1 AND gSkid_HR[IdxSkids_HR].Dosing_Pump_202.P202_HOA = 8 THEN
			gSkid_HR[IdxSkids_HR].VisBool.P202_MODE := 1;
		ELSE
			gSkid_HR[IdxSkids_HR].VisBool.P202_MODE := 0;
		END_IF;

		IF gSkid_HR[IdxSkids_HR].Pmax_General_Variables.SCREEN_LOCK = 1 AND gSkid_HR[IdxSkids_HR].Dosing_Pump_203.P203_HOA = 8 THEN
			gSkid_HR[IdxSkids_HR].VisBool.P203_MODE := 1;
		ELSE
			gSkid_HR[IdxSkids_HR].VisBool.P203_MODE := 0;
		END_IF;

		IF gSkid_HR[IdxSkids_HR].Pmax_General_Variables.SCREEN_LOCK = 1 AND gSkid_HR[IdxSkids_HR].Dosing_Pump_204.P204_HOA = 8 THEN
			gSkid_HR[IdxSkids_HR].VisBool.P204_MODE := 1;
		ELSE
			gSkid_HR[IdxSkids_HR].VisBool.P204_MODE := 0;
		END_IF;

		IF gSkid_HR[IdxSkids_HR].Pmax_General_Variables.UNIT_ID_DOSE = 0 THEN
			gSkid_HR[IdxSkids_HR].VisBool.IOSTATUS := 1;
		ELSE
			gSkid_HR[IdxSkids_HR].VisBool.IOSTATUS := 0;
		END_IF;

	END_FOR;

END_ACTION
```

#### Chart_Buffer.st
```iecst
ACTION Chart_Buffer:

	FOR IdxSkids_LR := 0 TO MAX_SKIDS_LR DO

		bufferIndex := 0;
		sampleTrigger := FALSE;

		samplingTimer(IN := NOT sampleTrigger, PT := T#1S);

		IF samplingTimer.Q THEN
			sampleTrigger := TRUE;
			samplingTimer(IN := FALSE);
		END_IF;

		IF sampleTrigger THEN
			sampleTrigger := FALSE;

			// Grab CD to store
			gSkid_LR[IdxSkids_LR].Sensor_Variables.CD101_BUFFER[bufferIndex] := gSkid_LR[IdxSkids_LR].Sensor_Variables.CD101

        	// Increment buffer index with wraparound
			bufferIndex := bufferIndex + 1;
			IF bufferIndex >= 600 THEN
				bufferIndex := 0;
			END_IF;

		END_IF;

	END_FOR;

END_ACTION
```

### Program Logical/Services (IEC)

#### Cyclic.st - Cyclic code
```iecst
PROGRAM _CYCLIC

	Services_Alarms_action;
	//Recipe_Action;

END_PROGRAM
```

#### Init.st - Init code
```iecst
PROGRAM _INIT

	//FOR IdxSkids_LR := 0 TO MAX_SKIDS_LR DO
	//	gSkid_LR[IdxSkids_LR].Notes.LOCATION := NOTES_LR[IdxSkids_LR];
	//END_FOR;

	IF DiagCpuIsARsim() OR DiagCpuIsSimulated() THEN
		gServices.DeviceName := 'USER_DEVICE_SIM';
	ELSE
		gServices.DeviceName :=  'USER_DEVICE';
	END_IF;

	//gServices.Alarms.Internal.MpAlarmXListUI_0.UISetup.AlarmListSize	:= 50;

	gSkid_LR[0].AlarmX_MpLink := gAlarmXCore_LR_0;
	gSkid_LR[1].AlarmX_MpLink := gAlarmXCore_LR_1;
	gSkid_LR[2].AlarmX_MpLink := gAlarmXCore_LR_2;
	gSkid_LR[3].AlarmX_MpLink := gAlarmXCore_LR_3;
	gSkid_LR[4].AlarmX_MpLink := gAlarmXCore_LR_4;
	gSkid_LR[5].AlarmX_MpLink := gAlarmXCore_LR_5;
	gSkid_LR[6].AlarmX_MpLink := gAlarmXCore_LR_6;
	gSkid_LR[7].AlarmX_MpLink := gAlarmXCore_LR_7;
	gSkid_LR[8].AlarmX_MpLink := gAlarmXCore_LR_8;
	gSkid_LR[9].AlarmX_MpLink := gAlarmXCore_LR_9;
	gSkid_LR[10].AlarmX_MpLink := gAlarmXCore_LR_10;
	gSkid_LR[11].AlarmX_MpLink := gAlarmXCore_LR_11;
	gSkid_LR[12].AlarmX_MpLink := gAlarmXCore_LR_12;
	gSkid_LR[13].AlarmX_MpLink := gAlarmXCore_LR_13;
	gSkid_LR[14].AlarmX_MpLink := gAlarmXCore_LR_14;
	gSkid_LR[15].AlarmX_MpLink := gAlarmXCore_LR_15;
	gSkid_LR[16].AlarmX_MpLink := gAlarmXCore_LR_16;
	gSkid_LR[17].AlarmX_MpLink := gAlarmXCore_LR_17;
	gSkid_LR[18].AlarmX_MpLink := gAlarmXCore_LR_18;
	gSkid_LR[19].AlarmX_MpLink := gAlarmXCore_LR_19;
	gSkid_LR[20].AlarmX_MpLink := gAlarmXCore_LR_20;
	gSkid_LR[21].AlarmX_MpLink := gAlarmXCore_LR_21;
	gSkid_LR[22].AlarmX_MpLink := gAlarmXCore_LR_22;
//	gSkid_LR[23].AlarmX_MpLink := gAlarmXCore_LR_23;
//	gSkid_LR[24].AlarmX_MpLink := gAlarmXCore_LR_24;
//	gSkid_LR[25].AlarmX_MpLink := gAlarmXCore_LR_25;

	gSkid_LR[0].AlarmXHistory_MpLink := gAlarmXHistory_LR_0;
	gSkid_LR[1].AlarmXHistory_MpLink := gAlarmXHistory_LR_1;
	gSkid_LR[2].AlarmXHistory_MpLink := gAlarmXHistory_LR_2;
	gSkid_LR[3].AlarmXHistory_MpLink := gAlarmXHistory_LR_3;
	gSkid_LR[4].AlarmXHistory_MpLink := gAlarmXHistory_LR_4;
	gSkid_LR[5].AlarmXHistory_MpLink := gAlarmXHistory_LR_5;
	gSkid_LR[6].AlarmXHistory_MpLink := gAlarmXHistory_LR_6;
	gSkid_LR[7].AlarmXHistory_MpLink := gAlarmXHistory_LR_7;
	gSkid_LR[8].AlarmXHistory_MpLink := gAlarmXHistory_LR_8;
	gSkid_LR[9].AlarmXHistory_MpLink := gAlarmXHistory_LR_9;
	gSkid_LR[10].AlarmXHistory_MpLink := gAlarmXHistory_LR_10;
	gSkid_LR[11].AlarmXHistory_MpLink := gAlarmXHistory_LR_11;
	gSkid_LR[12].AlarmXHistory_MpLink := gAlarmXHistory_LR_12;
	gSkid_LR[13].AlarmXHistory_MpLink := gAlarmXHistory_LR_13;
	gSkid_LR[14].AlarmXHistory_MpLink := gAlarmXHistory_LR_14;
	gSkid_LR[15].AlarmXHistory_MpLink := gAlarmXHistory_LR_15;
	gSkid_LR[16].AlarmXHistory_MpLink := gAlarmXHistory_LR_16;
	gSkid_LR[17].AlarmXHistory_MpLink := gAlarmXHistory_LR_17;
	gSkid_LR[18].AlarmXHistory_MpLink := gAlarmXHistory_LR_18;
	gSkid_LR[19].AlarmXHistory_MpLink := gAlarmXHistory_LR_19;
	gSkid_LR[20].AlarmXHistory_MpLink := gAlarmXHistory_LR_20;
	gSkid_LR[21].AlarmXHistory_MpLink := gAlarmXHistory_LR_21;
	gSkid_LR[22].AlarmXHistory_MpLink := gAlarmXHistory_LR_22;
	//	gSkid_LR[23].AlarmXHistory_MpLink := gAlarmXHistory_LR_23;
	//	gSkid_LR[24].AlarmXHistory_MpLink := gAlarmXHistory_LR_24;
	//	gSkid_LR[25].AlarmXHistory_MpLink := gAlarmXHistory_LR_25;

	gSkid_HR[0].AlarmX_MpLink := gAlarmXCore_HR_0;

END_PROGRAM
```

#### Exit.st - Exit code
```iecst
PROGRAM _EXIT

	FOR IdxSkids_LR := 0 TO MAX_SKIDS_LR DO
		gServices.Alarms_LR[IdxSkids_LR].Internal.MpAlarmXCore_0(MpLink := ADR(gSkid_LR[IdxSkids_LR].AlarmX_MpLink), Enable := FALSE);
		gServices.Alarms_LR[IdxSkids_LR].Internal.MpAlarmXListUI_0(MpLink := ADR(gSkid_LR[IdxSkids_LR].AlarmX_MpLink), Enable := FALSE);
		gServices.Alarms_LR[IdxSkids_LR].Internal.MpAlarmXHistory_0(MpLink := ADR(gSkid_LR[IdxSkids_LR].AlarmXHistory_MpLink), Enable := FALSE);
		gServices.Alarms_LR[IdxSkids_LR].Internal.MpAlarmXHistoryUI_0(MpLink := ADR(gSkid_LR[IdxSkids_LR].AlarmXHistory_MpLink), Enable := FALSE);
	END_FOR;

	FOR IdxSkids_HR := 0 TO MAX_SKIDS_HR DO
		gServices.Alarms_HR[IdxSkids_HR].Internal.MpAlarmXCore_0(MpLink := ADR(gSkid_HR[IdxSkids_HR].AlarmX_MpLink), Enable := FALSE);
		gServices.Alarms_HR[IdxSkids_HR].Internal.MpAlarmXListUI_0(MpLink := ADR(gSkid_HR[IdxSkids_HR].AlarmX_MpLink), Enable := FALSE);
//		gServices.Alarms_HR[IdxSkids_HR].Internal.MpAlarmXHistory_0(MpLink := ADR(gAlarmXHistory), Enable := FALSE);
//		gServices.Alarms_HR[IdxSkids_HR].Internal.MpAlarmXHistoryUI_0(MpLink := ADR(gAlarmXHistory), Enable := FALSE);
	END_FOR;

	gServices.Alarms_Global.MpAlarmXCore_0(Enable := FALSE);
	gServices.Alarms_Global.MpAlarmXListUI_0(Enable := FALSE);
	gServices.Alarms_Global.MpAlarmXHistory_0(Enable := FALSE);
	gServices.Alarms_Global.MpAlarmXHistoryUI_0(Enable := FALSE);

	gServices.Recipe.MpRecipeRegPar(Enable := FALSE);
	gServices.Recipe.MpRecipeXml(Enable := FALSE);

END_PROGRAM
```

#### Variables.var - Local variables
```iecst
VAR
	IdxSkids_LR : INT := 0;
	IdxAlarmsActive : INT := 0;
	IdxSkids_HR : INT := 0;
END_VAR
```

#### Alarms.st
```iecst
ACTION Services_Alarms_action:
//
//		// Case for handling the alarm history
//	CASE gServices.Alarms_LR[IdxSkids_LR].Internal.StateExportHistory OF
//		0:
//			IF gServices.Alarms_LR[IdxSkids_LR].In.ExportHistory THEN
//				HA_AlarmX_Helper(gSkid_LR[IdxSkids_LR].AlarmX_MpLink,'',HA_ALARMX_ACTION_LOG_ONLY,'HISTORY EXPORTED',FALSE);
//				gServices.Alarms_LR[IdxSkids_LR].In.ExportHistory 									:= FALSE;
//				gServices.Alarms_LR[IdxSkids_LR].Internal.MpAlarmXHistory_0.Export 				:= TRUE;
//				gServices.Alarms_LR[IdxSkids_LR].Internal.StateExportHistory 						:= 10;
//			ELSIF gServices.Alarms_LR[IdxSkids_LR].In.ClearHistory THEN
//				HA_AlarmX_Helper(gSkid_LR[IdxSkids_LR].AlarmX_MpLink,'',HA_ALARMX_ACTION_LOG_ONLY,'HISTORY CLEARED',FALSE);
//				gServices.Alarms_LR[IdxSkids_LR].In.ClearHistory 									:= FALSE;
//				MpAlarmXClearHistory(gAlarmXHistory);
//			END_IF;
//		10:
//			IF gServices.Alarms_LR[IdxSkids_LR].Internal.MpAlarmXHistory_0.CommandDone OR gServices.Alarms_LR[IdxSkids_LR].Internal.MpAlarmXHistory_0.Error THEN
//				gServices.Alarms_LR[IdxSkids_LR].Internal.MpAlarmXHistory_0.Export 				:= FALSE;
//				gServices.Alarms_LR[IdxSkids_LR].Internal.StateExportHistory 						:= 0;
//			END_IF;
//	END_CASE;
//
//	//	IF gMain.ErrorReset THEN
//	//		gServices.Alarms_LR[IdxSkids_LR].In.ResetAlarms 											:= TRUE;
//	//	END_IF;
//
//	// Case for handling the alarm resetting
//	CASE gServices.Alarms_LR[IdxSkids_LR].Internal.StateResetAlarms OF
//		0:
//			IF gServices.Alarms_LR[IdxSkids_LR].In.ResetAlarms OR gVis.Global.ErrorReset THEN
//				HA_AlarmX_Helper(gSkid_LR[IdxSkids_LR].AlarmX_MpLink,'',HA_ALARMX_ACTION_LOG_ONLY,'ACKNOWLEDGE ALL',FALSE);
//				gServices.Alarms_LR[IdxSkids_LR].In.ResetAlarms 									:= FALSE;
//				gVis.Alarms.Active.UIConnect.AcknowledgeAll 							:= TRUE;
//				gServices.Alarms_LR[IdxSkids_LR].Internal.CTON_ResetDelay(IN := FALSE);
//				gServices.Alarms_LR[IdxSkids_LR].Internal.StateResetAlarms 						:= 10;
//			END_IF;
//		10:
//			// give UI time to process the reset
//			IF gServices.Alarms_LR[IdxSkids_LR].Internal.CTON_ResetDelay.Q THEN
//				gServices.Alarms_LR[IdxSkids_LR].Internal.CTON_ResetDelay(IN := FALSE);
//				gServices.Alarms_LR[IdxSkids_LR].Internal.StateResetAlarms 						:= 0;
//				gVis.Global.ErrorReset := FALSE;
//			ELSE
//				gServices.Alarms_LR[IdxSkids_LR].Internal.CTON_ResetDelay(IN := TRUE, PT := T#250ms);
//			END_IF;
//	END_CASE;
//
//
//	FOR IdxSkids_HR := 0 TO MAX_SKIDS_HR DO
//
//		//Reset only Selected Skid Alarms
//		IF gVis.Main.In.AckAllAlarms_Skid_HR[IdxSkids_HR] THEN
//
//			FOR IdxAlarmsActive := 0 TO 49 DO
//				IF gVis.Alarms.Active.UIConnect.AlarmList.Code[IdxAlarmsActive] = gUnit_HR[IdxSkids_HR] THEN
//					MpAlarmXAcknowledgeID(gSkid_LR[IdxSkids_LR].AlarmX_MpLink,gVis.Alarms.Active.UIConnect.AlarmList.InstanceID[IdxAlarmsActive]);
//				ELSIF gVis.Alarms.Active.UIConnect.AlarmList.Code[IdxAlarmsActive] = 0 THEN
//					EXIT;
//				END_IF;
//			END_FOR;
//
//			gVis.Main.In.AckAllAlarms_Skid_HR[IdxSkids_HR] := FALSE;
//
//			gServices.Alarms_LR[IdxSkids_LR].Internal.Alarm_Set_Delay_HR[IdxSkids_HR].IN := TRUE;
//
//		END_IF;
//
//		IF gServices.Alarms_LR[IdxSkids_LR].Internal.Alarm_Set_Delay_HR[IdxSkids_HR].Q THEN
//			brsmemset(ADR(gServices.Alarms_LR[IdxSkids_LR].Internal.Alarms_State_HR[IdxSkids_HR]),0,SIZEOF(gServices.Alarms_LR[IdxSkids_LR].Internal.Alarms_State_HR[IdxSkids_HR]));
//			gServices.Alarms_LR[IdxSkids_LR].Internal.Alarm_Set_Delay_HR[IdxSkids_HR].IN := FALSE;
//		END_IF;
//
//		gServices.Alarms_LR[IdxSkids_LR].Internal.Alarm_Set_Delay_HR[IdxSkids_HR](PT := T#15s);
//
//	END_FOR;
//
//

	IF gVis.Alarms_Global.Active.AckAll THEN

		gVis.Alarms_Global.Active.UIConnect.AcknowledgeAll := TRUE;
		gVis.Alarms_Global.Active.AckAll := FALSE;

	END_IF;

	FOR IdxSkids_LR := 0 TO MAX_SKIDS_LR DO

		//		//Reset only Selected Skid Alarms
		IF gVis.Main.In.AckAllAlarms_Skid_LR[IdxSkids_LR] THEN

			gVis.Alarms_LR[IdxSkids_LR].Active.UIConnect.AcknowledgeAll := TRUE;
			gVis.Main.In.AckAllAlarms_Skid_LR[IdxSkids_LR] := FALSE;

			gServices.Alarms_LR[IdxSkids_LR].Internal.Alarm_Set_Delay.IN := TRUE;
		END_IF;

		IF gServices.Alarms_LR[IdxSkids_LR].Internal.Alarm_Set_Delay.Q THEN
			brsmemset(ADR(gServices.Alarms_LR[IdxSkids_LR].Internal.Alarms_State),0,SIZEOF(gServices.Alarms_LR[IdxSkids_LR].Internal.Alarms_State));
			gServices.Alarms_LR[IdxSkids_LR].Internal.Alarm_Set_Delay.IN := FALSE;
		END_IF;

		gServices.Alarms_LR[IdxSkids_LR].Internal.Alarm_Set_Delay(PT := T#15s);

		gServices.Alarms_LR[IdxSkids_LR].Out.BufferInfo.Address	:= ADR(gServices.Alarms_LR[IdxSkids_LR].In.AlarmList);
		gServices.Alarms_LR[IdxSkids_LR].Out.BufferInfo.Size		:= SIZEOF(gServices.Alarms_LR[IdxSkids_LR].In.AlarmList);

		gServices.Alarms_LR[IdxSkids_LR].Internal.HA_AlarmXCore_0(MpLink := gSkid_LR[IdxSkids_LR].AlarmX_MpLink, enable := TRUE, pBuffer := ADR(gServices.Alarms_LR[IdxSkids_LR].In.AlarmList), pOutputData := ADR(gAlarmAddData));
		gServices.Alarms_LR[IdxSkids_LR].Internal.MpAlarmXCore_0(MpLink := ADR(gSkid_LR[IdxSkids_LR].AlarmX_MpLink), Enable := TRUE, ErrorReset := gErrorReset);
		gServices.Alarms_LR[IdxSkids_LR].Internal.MpAlarmXListUI_0(MpLink := ADR(gSkid_LR[IdxSkids_LR].AlarmX_MpLink), Enable := TRUE, ErrorReset := gErrorReset, UIConnect := ADR(gVis.Alarms_LR[IdxSkids_LR].Active.UIConnect));
		gServices.Alarms_LR[IdxSkids_LR].Internal.MpAlarmXHistory_0(MpLink := ADR(gSkid_LR[IdxSkids_LR].AlarmXHistory_MpLink), Enable := TRUE, ErrorReset := gErrorReset,DeviceName := ADR(gServices.DeviceName));
		gServices.Alarms_LR[IdxSkids_LR].Internal.MpAlarmXHistoryUI_0(MpLink := ADR(gSkid_LR[IdxSkids_LR].AlarmXHistory_MpLink), Enable := TRUE, ErrorReset := gErrorReset, UIConnect := ADR(gVis.Alarms_LR[IdxSkids_LR].History.UIConnect));

		gVis.Alarms_LR[IdxSkids_LR].Active.UIConnect.AcknowledgeAll := FALSE;
	END_FOR

	gServices.Alarms_Global.HA_AlarmXCore_0(MpLink := gAlarmXCore_Global, enable := TRUE, pBuffer := ADR(gServices.Alarms_Global.AlarmList), pOutputData := ADR(gAlarmAddData_Global));
	gServices.Alarms_Global.MpAlarmXCore_0(MpLink := ADR(gAlarmXCore_Global), Enable := TRUE, ErrorReset := gErrorReset);
	gServices.Alarms_Global.MpAlarmXListUI_0(MpLink := ADR(gAlarmXCore_Global), Enable := TRUE, ErrorReset := gErrorReset, UIConnect := ADR(gVis.Alarms_Global.Active.UIConnect));

	gVis.Alarms_Global.Active.UIConnect.AcknowledgeAll := FALSE;

END_ACTION
```

#### Recipe.st
```iecst
ACTION Recipe_Action:

	IF gServices.Recipe.CreateNoteFile THEN
		gServices.Recipe.MpRecipeXml.Save := TRUE;
		IF gServices.Recipe.MpRecipeXml.CommandDone AND NOT gServices.Recipe.MpRecipeXml.Error THEN
			RecipeLoaded := TRUE;
			gServices.Recipe.MpRecipeXml.Save := FALSE;
			gServices.Recipe.CreateNoteFile := FALSE;

			FOR IdxSkids_LR := 0 TO MAX_SKIDS_LR DO
				gSkid_LR[IdxSkids_LR].Notes.LOCATION:= gRecipe_LR[IdxSkids_LR].Notes;
				gSkid_LR[IdxSkids_LR].RosterContact := gRecipe_LR[IdxSkids_LR].Contacts;
			END_FOR;

		END_IF
	END_IF

	IF NOT RecipeLoaded AND NOT gServices.Recipe.CreateNoteFile THEN
		gServices.Recipe.MpRecipeXml.Load := TRUE;
		IF gServices.Recipe.MpRecipeXml.CommandDone AND NOT gServices.Recipe.MpRecipeXml.Error THEN
			RecipeLoaded := TRUE;
			gServices.Recipe.MpRecipeXml.Load := FALSE;
			RECIPE_LR_TEMP := gRecipe_LR;

			FOR IdxSkids_LR := 0 TO MAX_SKIDS_LR DO
				gSkid_LR[IdxSkids_LR].Notes.LOCATION:= gRecipe_LR[IdxSkids_LR].Notes;
				gSkid_LR[IdxSkids_LR].RosterContact := gRecipe_LR[IdxSkids_LR].Contacts;
			END_FOR;

		ELSIF gServices.Recipe.MpRecipeXml.Error THEN
			gServices.Recipe.MpRecipeXml.Load := FALSE;
			gServices.Recipe.MpRecipeXml.ErrorReset := TRUE;
			gServices.Recipe.CreateNoteFile := TRUE;
		END_IF;
	END_IF;

	IF RecipeLoaded THEN
		FOR IdxSkids_LR := 0 TO MAX_SKIDS_LR DO
			gRecipe_LR[IdxSkids_LR].Notes := gSkid_LR[IdxSkids_LR].Notes.LOCATION;
			gRecipe_LR[IdxSkids_LR].Contacts := gSkid_LR[IdxSkids_LR].RosterContact;
		END_FOR;
	END_IF;

	IF brsmemcmp(ADR(gRecipe_LR),ADR(RECIPE_LR_TEMP),SIZEOF(RECIPE_LR_TEMP)) <> 0 AND RecipeLoaded THEN
		gServices.Recipe.MpRecipeXml.Save := TRUE;
		IF gServices.Recipe.MpRecipeXml.CommandDone AND NOT gServices.Recipe.MpRecipeXml.Error THEN
			gServices.Recipe.MpRecipeXml.Save := FALSE;
			RECIPE_LR_TEMP := gRecipe_LR;
		END_IF;
	END_IF;

	gServices.Recipe.MpRecipeRegPar(MpLink := ADR(gRecipeXml), Enable := TRUE, ErrorReset := gErrorReset, PVName := ADR('gRecipe_LR'));

	gServices.Recipe.MpRecipeXml(MpLink := ADR(gRecipeXml), Enable := TRUE, ErrorReset := gErrorReset, DeviceName := ADR('USER_DEVICE'), FileName := ADR('RECIPE.xml'));

END_ACTION
```

### Program Logical/Main (IEC)

#### Main.st - Init, cyclic, exit code
```iecst
PROGRAM _INIT

END_PROGRAM

PROGRAM _CYCLIC

	FOR IdxSkids := 0 TO MAX_SKIDS DO

		gSkid[IdxSkids].BufferTank.LI200P := (gSkid[IdxSkids].BufferTank.LI200 / BT_VOLUME)*100;

		// VISIBILITY TRIGGER SETTING. NEEDS TO BE MOVED TO VIS PROGRAM AT SOME POINT

		IF gSkid[IdxSkids].BufferTank.LSHH200 > LSHH200_TRIGGER THEN
			gSkid[IdxSkids].VisBool.LSHH200 := 1;
		ELSE
			gSkid[IdxSkids].VisBool.LSHH200 := 0;
		END_IF;

		IF gSkid[IdxSkids].Pmax_Pump_102.P102_LS > P102_LS_TRIGGER THEN
			gSkid[IdxSkids].VisBool.P102_LS := 1;
		ELSE
			gSkid[IdxSkids].VisBool.P102_LS := 0;
		END_IF;

		IF gSkid[IdxSkids].Pmax_Pump_103.P103_LS > P103_LS_TRIGGER THEN
			gSkid[IdxSkids].VisBool.P103_LS := 1;
		ELSE
			gSkid[IdxSkids].VisBool.P103_LS := 0;
		END_IF;

		IF gSkid[IdxSkids].Pmax_General_Variables.PMAX_HOA = 2 THEN
			gSkid[IdxSkids].VisBool.PMAX_MANUAL := 1;
		ELSE
			gSkid[IdxSkids].VisBool.PMAX_MANUAL := 0;
		END_IF;

		IF gSkid[IdxSkids].Dosing_Pump_201.P201_HOA = 0 OR gSkid[IdxSkids].Dosing_Pump_201.P201_HOA = 8  THEN
			gSkid[IdxSkids].VisBool.P201_PPM := 0;
		ELSE
			gSkid[IdxSkids].VisBool.P201_PPM := 1;
		END_IF;

		IF gSkid[IdxSkids].Dosing_Pump_202.P202_HOA = 0 OR gSkid[IdxSkids].Dosing_Pump_202.P202_HOA = 8  THEN
			gSkid[IdxSkids].VisBool.P202_PPM := 0;
		ELSE
			gSkid[IdxSkids].VisBool.P202_PPM := 1;
		END_IF;

		IF gSkid[IdxSkids].Dosing_Pump_203.P203_HOA = 0 OR gSkid[IdxSkids].Dosing_Pump_203.P203_HOA = 8  THEN
			gSkid[IdxSkids].VisBool.P203_PPM := 0;
		ELSE
			gSkid[IdxSkids].VisBool.P203_PPM := 1;
		END_IF;

		IF gSkid[IdxSkids].Dosing_Pump_201.P201_HOA = 8 THEN
			gSkid[IdxSkids].VisBool.P201_SP := 1;
		ELSE
			gSkid[IdxSkids].VisBool.P201_SP := 0;
		END_IF;

		IF gSkid[IdxSkids].Dosing_Pump_202.P202_HOA = 8 THEN
			gSkid[IdxSkids].VisBool.P202_SP := 1;
		ELSE
			gSkid[IdxSkids].VisBool.P202_SP := 0;
		END_IF;

		IF gSkid[IdxSkids].Dosing_Pump_203.P203_HOA = 8 THEN
			gSkid[IdxSkids].VisBool.P203_SP := 1;
		ELSE
			gSkid[IdxSkids].VisBool.P203_SP := 0;
		END_IF;

		IF gSkid[IdxSkids].Dosing_Pump_201.P201_PTYPE = 0 THEN
			gSkid[IdxSkids].VisBool.P201_DDA := 1;
			gSkid[IdxSkids].VisBool.P201_DME := 0;
		ELSE
			gSkid[IdxSkids].VisBool.P201_DDA := 0;
			gSkid[IdxSkids].VisBool.P201_DME := 1;
		END_IF;

		IF gSkid[IdxSkids].Dosing_Pump_201.P201_PTYPE = 0 AND gSkid[IdxSkids].Dosing_Pump_201.P201_XS = 1 THEN
			gSkid[IdxSkids].VisBool.P201_DDAGREEN := 1;
		ELSE
			gSkid[IdxSkids].VisBool.P201_DDAGREEN := 0;
		END_IF;

		IF gSkid[IdxSkids].Dosing_Pump_201.P201_PTYPE = 1 AND gSkid[IdxSkids].Dosing_Pump_201.P201_XS = 1 THEN
			gSkid[IdxSkids].VisBool.P201_DMEGREEN := 1;
		ELSE
			gSkid[IdxSkids].VisBool.P201_DMEGREEN := 0;
		END_IF;

		IF gSkid[IdxSkids].Dosing_Pump_201.P201_ENABLE = 1 THEN
			gSkid[IdxSkids].VisBool.P201_ENABLE_OPP := 0;
		ELSE
			gSkid[IdxSkids].VisBool.P201_ENABLE_OPP := 1;
		END_IF;

		IF gSkid[IdxSkids].Dosing_Pump_202.P202_ENABLE = 1 THEN
			gSkid[IdxSkids].VisBool.P202_ENABLE_OPP := 0;
		ELSE
			gSkid[IdxSkids].VisBool.P202_ENABLE_OPP := 1;
		END_IF;

		IF gSkid[IdxSkids].Dosing_Pump_203.P203_ENABLE = 1 THEN
			gSkid[IdxSkids].VisBool.P203_ENABLE_OPP := 0;
		ELSE
			gSkid[IdxSkids].VisBool.P203_ENABLE_OPP := 1;
		END_IF;

		IF gSkid[IdxSkids].Pmax_Pump_102.P102_WARN > 0 THEN
			gSkid[IdxSkids].VisBool.P102_WARN := 1;
		ELSE
			gSkid[IdxSkids].VisBool.P102_WARN := 0;
		END_IF;

		IF gSkid[IdxSkids].Pmax_Pump_102.P102_ALARM > 0 THEN
			gSkid[IdxSkids].VisBool.P102_ALARM := 1;
		ELSE
			gSkid[IdxSkids].VisBool.P102_ALARM := 0;
		END_IF;

		IF gSkid[IdxSkids].Pmax_Pump_103.P103_WARN > 0 THEN
			gSkid[IdxSkids].VisBool.P103_WARN := 1;
		ELSE
			gSkid[IdxSkids].VisBool.P103_WARN := 0;
		END_IF;

		IF gSkid[IdxSkids].Pmax_Pump_103.P103_ALARM > 0 THEN
			gSkid[IdxSkids].VisBool.P103_ALARM := 1;
		ELSE
			gSkid[IdxSkids].VisBool.P103_ALARM := 0;
		END_IF;

		IF gSkid[IdxSkids].Pmax_Pump_104.P104_WARN > 0 THEN
			gSkid[IdxSkids].VisBool.P104_WARN := 1;
		ELSE
			gSkid[IdxSkids].VisBool.P104_WARN := 0;
		END_IF;

		IF gSkid[IdxSkids].Pmax_Pump_104.P104_ALARM > 0 THEN
			gSkid[IdxSkids].VisBool.P104_ALARM := 1;
		ELSE
			gSkid[IdxSkids].VisBool.P104_ALARM := 0;
		END_IF;

		IF gSkid[IdxSkids].Dosing_Pump_201.P201_WARN > 0 THEN
			gSkid[IdxSkids].VisBool.P201_WARN := 1;
		ELSE
			gSkid[IdxSkids].VisBool.P201_WARN := 0;
		END_IF;

		IF gSkid[IdxSkids].Dosing_Pump_201.P201_ALARM > 0 THEN
			gSkid[IdxSkids].VisBool.P201_ALARM := 1;
		ELSE
			gSkid[IdxSkids].VisBool.P201_ALARM := 0;
		END_IF;

		IF gSkid[IdxSkids].Dosing_Pump_202.P202_WARN > 0 THEN
			gSkid[IdxSkids].VisBool.P202_WARN := 1;
		ELSE
			gSkid[IdxSkids].VisBool.P202_WARN := 0;
		END_IF;

		IF gSkid[IdxSkids].Dosing_Pump_202.P202_ALARM > 0 THEN
			gSkid[IdxSkids].VisBool.P202_ALARM := 1;
		ELSE
			gSkid[IdxSkids].VisBool.P202_ALARM := 0;
		END_IF;

		IF gSkid[IdxSkids].Dosing_Pump_203.P203_WARN > 0 THEN
			gSkid[IdxSkids].VisBool.P203_WARN := 1;
		ELSE
			gSkid[IdxSkids].VisBool.P203_WARN := 0;
		END_IF;

		IF gSkid[IdxSkids].Dosing_Pump_203.P203_ALARM > 0 THEN
			gSkid[IdxSkids].VisBool.P203_ALARM := 1;
		ELSE
			gSkid[IdxSkids].VisBool.P203_ALARM := 0;
		END_IF;

		IF gSkid[IdxSkids].Dosing_Pump_201.P201_ADJ = 1 AND gSkid[IdxSkids].VisBool.P201_PPM = 1 THEN
			gSkid[IdxSkids].VisBool.P201_APPM := 1;
		ELSE
			gSkid[IdxSkids].VisBool.P201_APPM := 0;
		END_IF;

		IF gSkid[IdxSkids].Dosing_Pump_202.P202_ADJ = 1 AND gSkid[IdxSkids].VisBool.P202_PPM = 1 THEN
			gSkid[IdxSkids].VisBool.P202_APPM := 1;
		ELSE
			gSkid[IdxSkids].VisBool.P202_APPM := 0;
		END_IF;

		IF gSkid[IdxSkids].Dosing_Pump_203.P203_ADJ = 1 AND gSkid[IdxSkids].VisBool.P203_PPM = 1 THEN
			gSkid[IdxSkids].VisBool.P203_APPM := 1;
		ELSE
			gSkid[IdxSkids].VisBool.P203_APPM := 0;
		END_IF;

		IF gSkid[IdxSkids].Sensor_Variables.FI301_MODE = 0 AND gSkid[IdxSkids].Pmax_General_Variables.SCREEN_LOCK = 1 THEN
			gSkid[IdxSkids].VisBool.FI301_MODE_OPP := 1;
		ELSE
			gSkid[IdxSkids].VisBool.FI301_MODE_OPP := 0;
		END_IF;

		IF gSkid[IdxSkids].Sensor_Variables.FI302_MODE = 0 AND gSkid[IdxSkids].Pmax_General_Variables.SCREEN_LOCK = 1 THEN
			gSkid[IdxSkids].VisBool.FI302_MODE_OPP := 1;
		ELSE
			gSkid[IdxSkids].VisBool.FI302_MODE_OPP := 0;
		END_IF;

		IF gSkid[IdxSkids].Sensor_Variables.FI303_MODE = 0 AND gSkid[IdxSkids].Pmax_General_Variables.SCREEN_LOCK = 1 THEN
			gSkid[IdxSkids].VisBool.FI303_MODE_OPP := 1;
		ELSE
			gSkid[IdxSkids].VisBool.FI303_MODE_OPP := 0;
		END_IF;

		IF gSkid[IdxSkids].Sensor_Variables.FI301_MODE = 1 AND gSkid[IdxSkids].Pmax_General_Variables.SCREEN_LOCK = 1 THEN
			gSkid[IdxSkids].VisBool.FI301_MODE := 1;
		ELSE
			gSkid[IdxSkids].VisBool.FI301_MODE := 0;
		END_IF;

		IF gSkid[IdxSkids].Sensor_Variables.FI302_MODE = 1 AND gSkid[IdxSkids].Pmax_General_Variables.SCREEN_LOCK = 1 THEN
			gSkid[IdxSkids].VisBool.FI302_MODE := 1;
		ELSE
			gSkid[IdxSkids].VisBool.FI302_MODE := 0;
		END_IF;

		IF gSkid[IdxSkids].Sensor_Variables.FI303_MODE = 1 AND gSkid[IdxSkids].Pmax_General_Variables.SCREEN_LOCK = 1 THEN
			gSkid[IdxSkids].VisBool.FI303_MODE := 1;
		ELSE
			gSkid[IdxSkids].VisBool.FI303_MODE := 0;
		END_IF;

		IF gSkid[IdxSkids].Sensor_Variables.XV101 = 0 AND gSkid[IdxSkids].Sensor_Variables.XV101_ENABLE = 1 THEN
			gSkid[IdxSkids].VisBool.XV101_OPP := 1;
		ELSE
			gSkid[IdxSkids].VisBool.XV101_OPP := 0;
		END_IF;

		IF gSkid[IdxSkids].Sensor_Variables.XV101 = 1 AND gSkid[IdxSkids].Sensor_Variables.XV101_ENABLE = 1 THEN
			gSkid[IdxSkids].VisBool.XV101 := 1;
		ELSE
			gSkid[IdxSkids].VisBool.XV101 := 0;
		END_IF;

		IF gSkid[IdxSkids].Sensor_Variables.XV102 = 1 THEN
			gSkid[IdxSkids].VisBool.XV102_OPP := 0;
		ELSE
			gSkid[IdxSkids].VisBool.XV102_OPP := 1;
		END_IF;

		IF gSkid[IdxSkids].Sensor_Variables.XV103 = 1 THEN
			gSkid[IdxSkids].VisBool.XV103_OPP := 0;
		ELSE
			gSkid[IdxSkids].VisBool.XV103_OPP := 1;
		END_IF;

		IF gSkid[IdxSkids].Sensor_Variables.XV104 = 1 THEN
			gSkid[IdxSkids].VisBool.XV104_OPP := 0;
		ELSE
			gSkid[IdxSkids].VisBool.XV104_OPP := 1;
		END_IF;

		IF gSkid[IdxSkids].Sensor_Variables.XV201 = 1 THEN
			gSkid[IdxSkids].VisBool.XV201_OPP := 0;
		ELSE
			gSkid[IdxSkids].VisBool.XV201_OPP := 1;
		END_IF;

		IF gSkid[IdxSkids].Sensor_Variables.XV202 = 1 THEN
			gSkid[IdxSkids].VisBool.XV202_OPP := 0;
		ELSE
			gSkid[IdxSkids].VisBool.XV202_OPP := 1;
		END_IF;

		IF gSkid[IdxSkids].Sensor_Variables.XV203 = 1 THEN
			gSkid[IdxSkids].VisBool.XV203_OPP := 0;
		ELSE
			gSkid[IdxSkids].VisBool.XV203_OPP := 1;
		END_IF;

		IF gSkid[IdxSkids].Dosing_Pump_201.P201_PTYPE = 1 THEN
			gSkid[IdxSkids].VisBool.P201_PTYPE_OPP := 0;
		ELSE
			gSkid[IdxSkids].VisBool.P201_PTYPE_OPP := 1;
		END_IF;

		IF gSkid[IdxSkids].Pmax_General_Variables.SCREEN_LOCK = 1 AND gSkid[IdxSkids].Pmax_General_Variables.PMAX_HOA = 2 THEN
			gSkid[IdxSkids].VisBool.P101_MODE := 1;
			gSkid[IdxSkids].VisBool.P102_MODE := 1;
			gSkid[IdxSkids].VisBool.P103_MODE := 1;
			gSkid[IdxSkids].VisBool.P104_MODE := 1;
		ELSE
			gSkid[IdxSkids].VisBool.P101_MODE := 0;
			gSkid[IdxSkids].VisBool.P102_MODE := 0;
			gSkid[IdxSkids].VisBool.P103_MODE := 0;
			gSkid[IdxSkids].VisBool.P104_MODE := 0;
		END_IF;

		IF gSkid[IdxSkids].Pmax_General_Variables.SCREEN_LOCK = 1 AND gSkid[IdxSkids].Dosing_Pump_201.P201_HOA = 8 THEN
			gSkid[IdxSkids].VisBool.P201_MODE := 1;
		ELSE
			gSkid[IdxSkids].VisBool.P201_MODE := 0;
		END_IF;

		IF gSkid[IdxSkids].Pmax_General_Variables.SCREEN_LOCK = 1 AND gSkid[IdxSkids].Dosing_Pump_202.P202_HOA = 8 THEN
			gSkid[IdxSkids].VisBool.P202_MODE := 1;
		ELSE
			gSkid[IdxSkids].VisBool.P202_MODE := 0;
		END_IF;

		IF gSkid[IdxSkids].Pmax_General_Variables.SCREEN_LOCK = 1 AND gSkid[IdxSkids].Dosing_Pump_203.P203_HOA = 8 THEN
			gSkid[IdxSkids].VisBool.P203_MODE := 1;
		ELSE
			gSkid[IdxSkids].VisBool.P203_MODE := 0;
		END_IF;

	END_FOR;

END_PROGRAM

PROGRAM _EXIT
	(* Insert code here *)

END_PROGRAM
```

#### Variables.var - Local variables
```iecst
VAR
	IdxSkids : INT;
	IdxAlarmsActive : INT;
	Client : httpsClient;
	IcmpPing_0 : IcmpPing;
	HostByName_0 : HostByName;
	JSON_Parsed : ARRAY[0..MAX_JSON_PARSE_PAIR_IDX] OF HA_JSON_Parse_Pair_typ;
	HA_JSON_Parse_0 : HA_JSON_Parse;
	IdxJSON : DINT;
	Authorization_Bearer : STRING[250];
	JSON_Parsed_UserInfo : ARRAY[0..MAX_JSON_PARSE_PAIR_IDX] OF HA_JSON_Parse_Pair_typ;
	HA_JSON_Parse_1 : HA_JSON_Parse;
	IdxClients : INT;
	ArUserCreate_0 : ArUserCreate;
	ArUserSetPassword_0 : ArUserSetPassword;
	Header : httpRequestHeader_t;
	API_Login_FB_0 : API_Login_FB;
END_VAR
```

#### API_Calls.st
```iecst
ACTION API_Calls_Action:

	Client.option 			:= httpOPTION_HTTP_11;
	Client.pHost 			:= ADR('cci-api-development-wjc4fopyua-uc.a.run.app');

	Header.protocol			:= 'HTTP/1.1';
	Header.host				:= 'cci-api-development-wjc4fopyua-uc.a.run.app';
	Header.contentType		:= 'application/json';
	Header.connection		:= 'keep-alive';
	Header.userLine[0].name	:= 'User-Agent';
	Header.userLine[0].value := 'SCADA';

	API_Login_FB_0(sUser := 'm.gogela@cleanchemi.com', sPassword := 'Fire1776', HttpClientRef := Client, RequestHeader := Header);

	//Post_Login_0(Client := Client,username := 'm.gogela@cleanchemi.com',password := 'Fire1776');

//	HA_JSON_Parse_0(pBuffer := ADR(Post_Login_0.ResponseData), pPairs := ADR(JSON_Parsed));

	FOR IdxJSON := 0 TO MAX_JSON_PARSE_PAIR_IDX DO
		IF JSON_Parsed[IdxJSON].Name = 'access' THEN
			brsmemcpy(ADR(Authorization_Bearer),ADR(JSON_Parsed[IdxJSON].Value)+1,LEN(JSON_Parsed[IdxJSON].Value)-2);
		END_IF;
	END_FOR;

	IcmpPing_0(pHost := ADR('google.com'), timeout := 10);

	HostByName_0(pName :=  ADR('cci-api-development-wjc4fopyua-uc.a.run.app'));

	//	GET_UserInfo_0(Client := Client, sAuthorization := Authorization_Bearer);

	//	HA_JSON_Parse_1(pBuffer := ADR(GET_UserInfo_0.ResponseData), pPairs := ADR(JSON_Parsed_UserInfo));

	FOR IdxClients := 0 TO MAX_CLIENTS DO

		IF gVis.Global.ClientInfo[IdxClients].LoginRequest THEN
			gVis.Global.ClientInfo[IdxClients].LoginSuccess := TRUE;
			gVis.Global.ClientInfo[IdxClients].LoginRequest := FALSE;
		END_IF;

	END_FOR;

	ArUserCreate_0();
	ArUserSetPassword_0();

END_ACTION
```

#### LocalFunctions.fun - not listed in the package file held
```iecst
{REDUND_ERROR} FUNCTION_BLOCK Post_Login (*TODO: Add your comment here*) (*$GROUP=User,$CAT=User,$GROUPICON=User.png,$CATICON=User.png*)
	VAR_INPUT
		username : STRING[80];
		password : STRING[80];
		bEnable : BOOL;
		bRequest : BOOL;
	END_VAR
	VAR_OUTPUT
		Phase : UINT;
		Status : {REDUND_UNREPLICABLE} UINT;
		ResponseStatus : {REDUND_UNREPLICABLE} STRING[280];
		Authorization : STRING[200];
		ResponseData : {REDUND_UNREPLICABLE} STRING[2000];
	END_VAR
	VAR_IN_OUT
		HttpClientRef : httpsClient;
	END_VAR
	VAR
		RequestHeader : {REDUND_UNREPLICABLE} httpRequestHeader_t;
		Host : {REDUND_UNREPLICABLE} STRING[80];
		ResponseHeader : {REDUND_UNREPLICABLE} httpResponseHeader_t;
		Ressource : {REDUND_UNREPLICABLE} STRING[80];
		sHeader : {REDUND_UNREPLICABLE} STRING[300];
		bEnabled : {REDUND_UNREPLICABLE} BOOL;
		RequestDataJson : {REDUND_UNREPLICABLE} STRING[1000];
	END_VAR
END_FUNCTION_BLOCK

{REDUND_ERROR} FUNCTION_BLOCK GET_UserInfo (*TODO: Add your comment here*) (*$GROUP=User,$CAT=User,$GROUPICON=User.png,$CATICON=User.png*)
	VAR_INPUT
		sAuthorization : STRING[250];
		bEnable : BOOL;
		bRequest : BOOL;
	END_VAR
	VAR_OUTPUT
		Phase : UINT;
		Status : {REDUND_UNREPLICABLE} UINT;
		ResponseStatus : {REDUND_UNREPLICABLE} STRING[280];
		ResponseData : {REDUND_UNREPLICABLE} STRING[2000];
	END_VAR
	VAR_IN_OUT
		HttpClientRef : httpsClient;
	END_VAR
	VAR
		RequestHeader : {REDUND_UNREPLICABLE} httpRequestHeader_t;
		Host : {REDUND_UNREPLICABLE} STRING[80];
		ResponseHeader : {REDUND_UNREPLICABLE} httpResponseHeader_t;
		Ressource : {REDUND_UNREPLICABLE} STRING[80];
		sHeader : {REDUND_UNREPLICABLE} STRING[400];
		bEnabled : {REDUND_UNREPLICABLE} BOOL;
		RequestDataJson : {REDUND_UNREPLICABLE} STRING[1000];
	END_VAR
END_FUNCTION_BLOCK
```

#### Alarms.st - not listed in the package file held
```iecst
ACTION Alarms_action:

	//SP Alarm
	IF gSkid[IdxSkids].Dosing_Alarms.DOSE_ALARM.0 THEN

	END_IF;

END_ACTION
```

#### GET_UserInfo.st - not listed in the package file held
```iecst
(* TODO: Add your comment here *)
FUNCTION_BLOCK GET_UserInfo

	IF bEnable AND NOT bEnabled THEN
		bEnabled	:= TRUE;
		sHeader		:= CONCAT('Authorization: Bearer ',sAuthorization);
		Ressource	:= '/auth/users/me/';
		Host		:= 'cci-api-development-wjc4fopyua-uc.a.run.app';

		HttpClientRef.option 			:= httpOPTION_HTTP_11;
		HttpClientRef.pHost 			:= ADR(Host);
		HttpClientRef.method 			:= httpMETHOD_GET;
		HttpClientRef.pUri 				:= ADR(Ressource);
		HttpClientRef.pRequestHeader	:= ADR(RequestHeader);
		HttpClientRef.pRequestData		:= ADR(RequestDataJson);
		HttpClientRef.requestDataLen	:= LEN(RequestDataJson);
		HttpClientRef.pResponseHeader	:= ADR(ResponseHeader);
		HttpClientRef.pResponseData 	:= ADR(ResponseData);
		HttpClientRef.responseDataSize	:= SIZEOF(ResponseData);

		RequestHeader.protocol			:= 'HTTP/1.1';
		RequestHeader.host				:= Host;
		RequestHeader.contentType		:= 'application/json';
		RequestHeader.contentLength		:=  LEN(RequestDataJson);
		RequestHeader.connection		:= 'keep-alive';
		RequestHeader.rawHeader.dataLen	:= LEN(sHeader);
		RequestHeader.rawHeader.pData	:= ADR(sHeader);
	//	RequestHeader.userLine[0].name	:= 'Authorization';
	//	RequestHeader.userLine[0].value := CONCAT('Bearer ','eyJhbGciOiJIUzI1NiIsInR5cCI6IkpXVCJ9.eyJ0b2tlbl90eXBlIjoiYWNjZXNzIiwiZXhwIjoxNzQ5MDYwOTYzLCJqdGkiOiJkNDg0MDAxMjM0MmE0YjJjYjQ2NzMwYjVhNGY1YTFmNyIsInVzZXJfaWQiOjEwfQ.AVaWOw9VqAKLQE9KLkQGM_h3jkvgIiEIJNefHxd0ypA');
		RequestHeader.userLine[1].name	:= 'User-Agent';
		RequestHeader.userLine[1].value := 'SCADA';

	ELSIF bEnable AND bEnabled THEN
		HttpClientRef.enable	:= TRUE;
		IF bRequest THEN
			HttpClientRef.send	:= TRUE;
		END_IF
	ELSIF NOT bEnable AND bEnabled THEN
		bEnabled	:= FALSE;
		bRequest	:= FALSE;
		HttpClientRef.enable	:= FALSE;
		HttpClientRef.send	:= FALSE;
	END_IF

	HttpClientRef();

	Status := HttpClientRef.status;
	Phase := HttpClientRef.phase;
	ResponseStatus := ResponseHeader.status;

END_FUNCTION_BLOCK
```

#### Post_Login.st - not listed in the package file held
```iecst
(* TODO: Add your comment here *)
FUNCTION_BLOCK Post_Login

	IF bEnable AND NOT bEnabled THEN
		bEnabled	:= TRUE;
		sHeader		:= '';
		Ressource	:= '/auth/jwt/create';
		Host		:= 'cci-api-development-wjc4fopyua-uc.a.run.app';
		//sHeader		:= CONCAT('Authorization: ',sAuthorization);
		RequestDataJson :='{"username":"m.gogela@cleanchemi.com","password":"Fire1776"}';

		HttpClientRef.option 			:= httpOPTION_HTTP_11;
		HttpClientRef.pHost 			:= ADR(Host);
		HttpClientRef.method 			:= httpMETHOD_POST;
		HttpClientRef.pUri 				:= ADR(Ressource);
		HttpClientRef.pRequestHeader	:= ADR(RequestHeader);
		HttpClientRef.pRequestData		:= ADR(RequestDataJson);
		HttpClientRef.requestDataLen	:= LEN(RequestDataJson)+2; //According to WireShark there is a /r/n in the packet that is not being accounted for which requires us to add 2 bytes to the length
		HttpClientRef.pResponseHeader	:= ADR(ResponseHeader);
		HttpClientRef.pResponseData 	:= ADR(ResponseData);
		HttpClientRef.responseDataSize	:= SIZEOF(ResponseData);

		RequestHeader.protocol			:= 'HTTP/1.1';
		RequestHeader.host				:= Host;
		RequestHeader.contentType		:= 'application/json';
		RequestHeader.contentLength		:=  LEN(RequestDataJson)+2; //According to WireShark there is a /r/n in the packet that is not being accounted for which requires us to add 2 bytes to the length
		RequestHeader.connection		:= 'keep-alive';
		//RequestHeader.userLine[0].name	:= 'Accept';
		//RequestHeader.userLine[0].value	:= '*/*';
		RequestHeader.rawHeader.dataLen	:= LEN(sHeader);
		RequestHeader.rawHeader.pData	:= ADR(sHeader);

	ELSIF bEnable AND bEnabled THEN
		HttpClientRef.enable	:= TRUE;
		IF bRequest THEN
			HttpClientRef.send	:= TRUE;
		END_IF
	ELSIF NOT bEnable AND bEnabled THEN
		bEnabled	:= FALSE;
		bRequest	:= FALSE;
		HttpClientRef.enable	:= FALSE;
		HttpClientRef.send	:= FALSE;
	END_IF

	HttpClientRef();

	Status := HttpClientRef.status;
	Phase := HttpClientRef.phase;
	ResponseStatus := ResponseHeader.status;

END_FUNCTION_BLOCK
```

### Program Logical/ModbusDriver

#### Variables.var
```iecst
VAR
	IdxModbusBlocks : USINT;
	ModbusDelay_TON : ARRAY[0..MAX_MODBUS_BLOCKS] OF TON;
END_VAR
```

#### Main.st
```iecst
PROGRAM _INIT

	gModbusDriver[0].BlockSend := TRUE;

END_PROGRAM

PROGRAM _CYCLIC

	IF gModbusDriver[IdxModbusBlocks].BlockRecieved THEN
		gModbusDriver[IdxModbusBlocks].BlockSend := FALSE;
		ModbusDelay_TON[IdxModbusBlocks].IN := TRUE;
	ELSIF NOT ModbusDelay_TON[IdxModbusBlocks].IN THEN
		gModbusDriver[IdxModbusBlocks].BlockSend := TRUE;
	END_IF;

	IF IdxModbusBlocks < MAX_MODBUS_BLOCKS AND ModbusDelay_TON[IdxModbusBlocks].Q THEN
		IdxModbusBlocks := IdxModbusBlocks + 1;
		ModbusDelay_TON[IdxModbusBlocks].IN := FALSE;
	ELSIF  ModbusDelay_TON[IdxModbusBlocks].Q THEN
		ModbusDelay_TON[IdxModbusBlocks].IN := FALSE;
		IdxModbusBlocks := 0;
	END_IF;

	ModbusDelay_TON[IdxModbusBlocks](PT := T#10ms);

END_PROGRAM

PROGRAM _EXIT
	(* Insert code here *)

END_PROGRAM
```

Listed in the project but not available here: Logical/Vis.typ, Logical/Process.typ, Logical/Libraries/Str2DtPvdr/Types.typ, Logical/Libraries/Str2DtPvdr/Constants.var, Logical/Libraries/HA_IO/Constants.var, Logical/Libraries/HA/Constants.var, Logical/Libraries/HA_Version/Constants.var, Logical/Libraries/HA_Convert/Constants.var, Logical/Libraries/HA_RAND/Types.typ, Logical/Libraries/HA_RAND/Constants.var, Logical/Libraries/HA_Array/Types.typ, Logical/Libraries/HA_SysErr/Constants.var, Logical/Libraries/HA_Str/Constants.var, Logical/Libraries/API_Login/Types.typ, Logical/Libraries/API_Login/Constants.var, Logical/Libraries/HA_Recipe/Constants.var, Logical/Libraries/HA_Sim/Constants.var, Logical/modbusTCP/IDEC_Real/Types.typ, Logical/modbusTCP/IDEC_Strng/Types.typ, Logical/modbusTCP/IDEC_Strng/Constants.var, Logical/modbusTCP/ModMaster/ModMaster.typ, Logical/modbusTCP/ModMaster_LR/ModMaster.typ, Logical/Services/Types.typ, Logical/Main/Types.typ
